        Win32ErrorCodeDescription := 'The password is too complex to be converted to a LAN Manager password. The LAN Manager password returned is a NULL string.';
    Win32ErrorCodes.ERROR_UNKNOWN_REVISION:
        Win32ErrorCodeDescription := 'The revision level is unknown.';
    Win32ErrorCodes.ERROR_REVISION_MISMATCH:
        Win32ErrorCodeDescription := 'Indicates two revision levels are incompatible.';
    Win32ErrorCodes.ERROR_INVALID_OWNER:
        Win32ErrorCodeDescription :=
            'This security ID may not be assigned as the owner of this object.';
    Win32ErrorCodes.ERROR_INVALID_PRIMARY_GROUP:
        Win32ErrorCodeDescription :=
            'This security ID may not be assigned as the primary group of an object.';
    Win32ErrorCodes.ERROR_NO_IMPERSONATION_TOKEN:
        Win32ErrorCodeDescription := 'An attempt has been made to operate on an impersonation token by a thread that is not currently impersonating a client.';
    Win32ErrorCodes.ERROR_CANT_DISABLE_MANDATORY:
        Win32ErrorCodeDescription := 'The group may not be disabled.';
    Win32ErrorCodes.ERROR_NO_LOGON_SERVERS:
        Win32ErrorCodeDescription :=
            'There are currently no logon servers available to service the logon request.';
    Win32ErrorCodes.ERROR_NO_SUCH_LOGON_SESSION:
        Win32ErrorCodeDescription :=
            'A specified logon session does not exist. It may already have been terminated.';
    Win32ErrorCodes.ERROR_NO_SUCH_PRIVILEGE:
        Win32ErrorCodeDescription := 'A specified privilege does not exist.';
    Win32ErrorCodes.ERROR_PRIVILEGE_NOT_HELD:
        Win32ErrorCodeDescription := 'A required privilege is not held by the client.';
    Win32ErrorCodes.ERROR_INVALID_ACCOUNT_NAME:
        Win32ErrorCodeDescription := 'The name provided is not a properly formed account name.';
    Win32ErrorCodes.ERROR_USER_EXISTS:
        Win32ErrorCodeDescription := 'The specified user already exists.';
    Win32ErrorCodes.ERROR_NO_SUCH_USER:
        Win32ErrorCodeDescription := 'The specified user does not exist.';
    Win32ErrorCodes.ERROR_GROUP_EXISTS:
        Win32ErrorCodeDescription := 'The specified group already exists.';
    Win32ErrorCodes.ERROR_NO_SUCH_GROUP:
        Win32ErrorCodeDescription := 'The specified group does not exist.';
    Win32ErrorCodes.ERROR_MEMBER_IN_GROUP:
        Win32ErrorCodeDescription := 'Either the specified user account is already a member of the specified group, or the specified group cannot be deleted because it contains a member.';
    Win32ErrorCodes.ERROR_MEMBER_NOT_IN_GROUP:
        Win32ErrorCodeDescription :=
            'The specified user account is not a member of the specified group account.';
    Win32ErrorCodes.ERROR_LAST_ADMIN:
        Win32ErrorCodeDescription :=
            'The last remaining administration account cannot be disabled or deleted.';
    Win32ErrorCodes.ERROR_WRONG_PASSWORD:
        Win32ErrorCodeDescription :=
            'Unable to update the password. The value provided as the current password is incorrect.';
    Win32ErrorCodes.ERROR_ILL_FORMED_PASSWORD:
        Win32ErrorCodeDescription := 'Unable to update the password. The value provided for the new password contains values that are not allowed in passwords.';
    Win32ErrorCodes.ERROR_PASSWORD_RESTRICTION:
        Win32ErrorCodeDescription := 'Unable to update the password. The value provided for the new password does not meet the length, complexity, or history requirement of the domain.';
    Win32ErrorCodes.ERROR_LOGON_FAILURE:
        Win32ErrorCodeDescription := 'Logon failure: unknown user name or bad password.';
    Win32ErrorCodes.ERROR_ACCOUNT_RESTRICTION:
        Win32ErrorCodeDescription := 'Logon failure: user account restriction.';
    Win32ErrorCodes.ERROR_INVALID_LOGON_HOURS:
        Win32ErrorCodeDescription := 'Logon failure: account logon time restriction violation.';
    Win32ErrorCodes.ERROR_INVALID_WORKSTATION:
        Win32ErrorCodeDescription := 'Logon failure: user not allowed to log on to this computer.';
    Win32ErrorCodes.ERROR_PASSWORD_EXPIRED:
        Win32ErrorCodeDescription := 'Logon failure: the specified account password has expired.';
    Win32ErrorCodes.ERROR_ACCOUNT_DISABLED:
        Win32ErrorCodeDescription := 'Logon failure: account currently disabled.';
    Win32ErrorCodes.ERROR_NONE_MAPPED:
        Win32ErrorCodeDescription := 'No mapping between account names and security IDs was done.';
    Win32ErrorCodes.ERROR_TOO_MANY_LUIDS_REQUESTED:
        Win32ErrorCodeDescription :=
            'Too many local user identifiers (LUIDs) were requested at one time.';
    Win32ErrorCodes.ERROR_LUIDS_EXHAUSTED:
        Win32ErrorCodeDescription := 'No more local user identifiers (LUIDs) are available.';
    Win32ErrorCodes.ERROR_INVALID_SUB_AUTHORITY:
        Win32ErrorCodeDescription :=
            'The subauthority part of a security ID is invalid for this particular use.';
    Win32ErrorCodes.ERROR_INVALID_ACL:
        Win32ErrorCodeDescription := 'The access control list (ACL) structure is invalid.';
    Win32ErrorCodes.ERROR_INVALID_SID:
        Win32ErrorCodeDescription := 'The security ID structure is invalid.';
    Win32ErrorCodes.ERROR_INVALID_SECURITY_DESCR:
        Win32ErrorCodeDescription := 'The security descriptor structure is invalid.';
    Win32ErrorCodes.ERROR_BAD_INHERITANCE_ACL:
        Win32ErrorCodeDescription :=
            'The inherited access control list (ACL) or access control entry (ACE) could not be built.';
    Win32ErrorCodes.ERROR_SERVER_DISABLED:
        Win32ErrorCodeDescription := 'The server is currently disabled.';
    Win32ErrorCodes.ERROR_SERVER_NOT_DISABLED:
        Win32ErrorCodeDescription := 'The server is currently enabled.';
    Win32ErrorCodes.ERROR_INVALID_ID_AUTHORITY:
        Win32ErrorCodeDescription :=
            'The value provided was an invalid value for an identifier authority.';
    Win32ErrorCodes.ERROR_ALLOTTED_SPACE_EXCEEDED:
        Win32ErrorCodeDescription :=
            'No more memory is available for security information updates.';
    Win32ErrorCodes.ERROR_INVALID_GROUP_ATTRIBUTES:
        Win32ErrorCodeDescription := 'The specified attributes are invalid, or incompatible with the attributes for the group as a whole.';
    Win32ErrorCodes.ERROR_BAD_IMPERSONATION_LEVEL:
        Win32ErrorCodeDescription := 'Either a required impersonation level was not provided, or the provided impersonation level is invalid.';
    Win32ErrorCodes.ERROR_CANT_OPEN_ANONYMOUS:
        Win32ErrorCodeDescription := 'Cannot open an anonymous level security token.';
    Win32ErrorCodes.ERROR_BAD_VALIDATION_CLASS:
        Win32ErrorCodeDescription := 'The validation information class requested was invalid.';
    Win32ErrorCodes.ERROR_BAD_TOKEN_TYPE:
        Win32ErrorCodeDescription :=
            'The type of the token is inappropriate for its attempted use.';
    Win32ErrorCodes.ERROR_NO_SECURITY_ON_OBJECT:
        Win32ErrorCodeDescription :=
            'Unable to perform a security operation on an object that has no associated security.';
    Win32ErrorCodes.ERROR_CANT_ACCESS_DOMAIN_INFO:
        Win32ErrorCodeDescription := 'Configuration information could not be read from the domain controller, either because the machine is unavailable, or access has been denied.';
    Win32ErrorCodes.ERROR_INVALID_SERVER_STATE:
        Win32ErrorCodeDescription := 'The security account manager (SAM) or local security authority (LSA) server was in the wrong state to perform the security operation.';
    Win32ErrorCodes.ERROR_INVALID_DOMAIN_STATE:
        Win32ErrorCodeDescription :=
            'The domain was in the wrong state to perform the security operation.';
    Win32ErrorCodes.ERROR_INVALID_DOMAIN_ROLE:
        Win32ErrorCodeDescription :=
            'This operation is only allowed for the Primary Domain Controller of the domain.';
    Win32ErrorCodes.ERROR_NO_SUCH_DOMAIN:
        Win32ErrorCodeDescription :=
            'The specified domain either does not exist or could not be contacted.';
    Win32ErrorCodes.ERROR_DOMAIN_EXISTS:
        Win32ErrorCodeDescription := 'The specified domain already exists.';
    Win32ErrorCodes.ERROR_DOMAIN_LIMIT_EXCEEDED:
        Win32ErrorCodeDescription :=
            'An attempt was made to exceed the limit on the number of domains per server.';
    Win32ErrorCodes.ERROR_INTERNAL_DB_CORRUPTION:
        Win32ErrorCodeDescription := 'Unable to complete the requested operation because of either a catastrophic media failure or a data structure corruption on the disk.';
    Win32ErrorCodes.ERROR_INTERNAL_ERROR:
        Win32ErrorCodeDescription := 'An internal error occurred.';
    Win32ErrorCodes.ERROR_GENERIC_NOT_MAPPED:
        Win32ErrorCodeDescription := 'Generic access types were contained in an access mask which should already be mapped to nongeneric types.';
    Win32ErrorCodes.ERROR_BAD_DESCRIPTOR_FORMAT:
        Win32ErrorCodeDescription :=
            'A security descriptor is not in the right format (absolute or self-relative).';
    Win32ErrorCodes.ERROR_NOT_LOGON_PROCESS:
        Win32ErrorCodeDescription := 'The requested action is restricted for use by logon processes only. The calling process has not registered as a logon process.';
    Win32ErrorCodes.ERROR_LOGON_SESSION_EXISTS:
        Win32ErrorCodeDescription :=
            'Cannot start a new logon session with an ID that is already in use.';
    Win32ErrorCodes.ERROR_NO_SUCH_PACKAGE:
        Win32ErrorCodeDescription := 'A specified authentication package is unknown.';
    Win32ErrorCodes.ERROR_BAD_LOGON_SESSION_STATE:
        Win32ErrorCodeDescription :=
            'The logon session is not in a state that is consistent with the requested operation.';
    Win32ErrorCodes.ERROR_LOGON_SESSION_COLLISION:
        Win32ErrorCodeDescription := 'The logon session ID is already in use.';
    Win32ErrorCodes.ERROR_INVALID_LOGON_TYPE:
        Win32ErrorCodeDescription := 'A logon request contained an invalid logon type value.';
    Win32ErrorCodes.ERROR_CANNOT_IMPERSONATE:
        Win32ErrorCodeDescription :=
            'Unable to impersonate using a named pipe until data has been read from that pipe.';
    Win32ErrorCodes.ERROR_RXACT_INVALID_STATE:
        Win32ErrorCodeDescription :=
            'The transaction state of a registry subtree is incompatible with the requested operation.';
    Win32ErrorCodes.ERROR_RXACT_COMMIT_FAILURE:
        Win32ErrorCodeDescription :=
            'An internal security database corruption has been encountered.';
    Win32ErrorCodes.ERROR_SPECIAL_ACCOUNT:
        Win32ErrorCodeDescription := 'Cannot perform this operation on built-in accounts.';
    Win32ErrorCodes.ERROR_SPECIAL_GROUP:
        Win32ErrorCodeDescription :=
            'Cannot perform this operation on this built-in special group.';
    Win32ErrorCodes.ERROR_SPECIAL_USER:
        Win32ErrorCodeDescription :=
            'Cannot perform this operation on this built-in special user.';
    Win32ErrorCodes.ERROR_MEMBERS_PRIMARY_GROUP:
        Win32ErrorCodeDescription := 'The user cannot be removed from a group because the group is currently the users primary group.';
    Win32ErrorCodes.ERROR_TOKEN_ALREADY_IN_USE:
        Win32ErrorCodeDescription := 'The token is already in use as a primary token.';
    Win32ErrorCodes.ERROR_NO_SUCH_ALIAS:
        Win32ErrorCodeDescription := 'The specified local group does not exist.';
    Win32ErrorCodes.ERROR_MEMBER_NOT_IN_ALIAS:
        Win32ErrorCodeDescription :=
            'The specified account name is not a member of the local group.';
    Win32ErrorCodes.ERROR_MEMBER_IN_ALIAS:
        Win32ErrorCodeDescription :=
            'The specified account name is already a member of the local group.';
    Win32ErrorCodes.ERROR_ALIAS_EXISTS:
        Win32ErrorCodeDescription := 'The specified local group already exists.';
    Win32ErrorCodes.ERROR_LOGON_NOT_GRANTED:
        Win32ErrorCodeDescription :=
            'Logon failure: the user has not been granted the requested logon type at this computer.';
    Win32ErrorCodes.ERROR_TOO_MANY_SECRETS:
        Win32ErrorCodeDescription :=
            'The maximum number of secrets that may be stored in a single system has been exceeded.';
    Win32ErrorCodes.ERROR_SECRET_TOO_LONG:
        Win32ErrorCodeDescription := 'The length of a secret exceeds the maximum length allowed.';
    Win32ErrorCodes.ERROR_INTERNAL_DB_ERROR:
        Win32ErrorCodeDescription :=
            'The local security authority database contains an internal inconsistency.';
    Win32ErrorCodes.ERROR_TOO_MANY_CONTEXT_IDS:
        Win32ErrorCodeDescription :=
            'During a logon attempt, the users security context accumulated too many security IDs.';
    Win32ErrorCodes.ERROR_LOGON_TYPE_NOT_GRANTED:
        Win32ErrorCodeDescription :=
            'Logon failure: the user has not been granted the requested logon type at this computer.';
    Win32ErrorCodes.ERROR_NT_CROSS_ENCRYPTION_REQUIRED:
        Win32ErrorCodeDescription :=
            'A cross-encrypted password is necessary to change a user password.';
    Win32ErrorCodes.ERROR_NO_SUCH_MEMBER:
        Win32ErrorCodeDescription := 'A new member could not be added to or removed from the local group because the member does not exist.';
    Win32ErrorCodes.ERROR_INVALID_MEMBER:
        Win32ErrorCodeDescription := 'A new member could not be added to a local group because the member has the wrong account type.';
    Win32ErrorCodes.ERROR_TOO_MANY_SIDS:
        Win32ErrorCodeDescription := 'Too many security IDs have been specified.';
    Win32ErrorCodes.ERROR_LM_CROSS_ENCRYPTION_REQUIRED:
        Win32ErrorCodeDescription :=
            'A cross-encrypted password is necessary to change this user password.';
    Win32ErrorCodes.ERROR_NO_INHERITANCE:
        Win32ErrorCodeDescription := 'Indicates an ACL contains no inheritable components.';
    Win32ErrorCodes.ERROR_FILE_CORRUPT:
        Win32ErrorCodeDescription := 'The file or directory is corrupted and unreadable.';
    Win32ErrorCodes.ERROR_DISK_CORRUPT:
        Win32ErrorCodeDescription := 'The disk structure is corrupted and unreadable.';
    Win32ErrorCodes.ERROR_NO_USER_SESSION_KEY:
        Win32ErrorCodeDescription :=
            'There is no user session key for the specified logon session.';
    Win32ErrorCodes.ERROR_LICENSE_QUOTA_EXCEEDED:
        Win32ErrorCodeDescription := 'The service being accessed is licensed for a particular number of connections. No more connections can be made to the service at this time because there are already as many connections as the service can accept.';
    Win32ErrorCodes.ERROR_WRONG_TARGET_NAME:
        Win32ErrorCodeDescription := 'Logon Failure: The target account name is incorrect.';
    Win32ErrorCodes.ERROR_MUTUAL_AUTH_FAILED:
        Win32ErrorCodeDescription := 'Mutual Authentication failed. The servers password is out of date at the domain controller.';
    Win32ErrorCodes.ERROR_TIME_SKEW:
        Win32ErrorCodeDescription := 'There is a time difference between the client and server.';
    Win32ErrorCodes.ERROR_CURRENT_DOMAIN_NOT_ALLOWED:
        Win32ErrorCodeDescription := 'This operation can not be performed on the current domain.';
    Win32ErrorCodes.ERROR_INVALID_WINDOW_HANDLE:
        Win32ErrorCodeDescription := 'Invalid window handle.';
    Win32ErrorCodes.ERROR_INVALID_MENU_HANDLE:
        Win32ErrorCodeDescription := 'Invalid menu handle.';
    Win32ErrorCodes.ERROR_INVALID_CURSOR_HANDLE:
        Win32ErrorCodeDescription := 'Invalid cursor handle.';
    Win32ErrorCodes.ERROR_INVALID_ACCEL_HANDLE:
        Win32ErrorCodeDescription := 'Invalid accelerator table handle.';
    Win32ErrorCodes.ERROR_INVALID_HOOK_HANDLE:
        Win32ErrorCodeDescription := 'Invalid hook handle.';
    Win32ErrorCodes.ERROR_INVALID_DWP_HANDLE:
        Win32ErrorCodeDescription := 'Invalid handle to a multiple-window position structure.';
    Win32ErrorCodes.ERROR_TLW_WITH_WSCHILD:
        Win32ErrorCodeDescription := 'Cannot create a top-level child window.';
    Win32ErrorCodes.ERROR_CANNOT_FIND_WND_CLASS:
        Win32ErrorCodeDescription := 'Cannot find window class.';
    Win32ErrorCodes.ERROR_WINDOW_OF_OTHER_THREAD:
        Win32ErrorCodeDescription := 'Invalid window; it belongs to other thread.';
    Win32ErrorCodes.ERROR_HOTKEY_ALREADY_REGISTERED:
        Win32ErrorCodeDescription := 'Hot key is already registered.';
    Win32ErrorCodes.ERROR_CLASS_ALREADY_EXISTS:
        Win32ErrorCodeDescription := 'Class already exists.';
    Win32ErrorCodes.ERROR_CLASS_DOES_NOT_EXIST:
        Win32ErrorCodeDescription := 'Class does not exist.';
    Win32ErrorCodes.ERROR_CLASS_HAS_WINDOWS:
        Win32ErrorCodeDescription := 'Class still has open windows.';
    Win32ErrorCodes.ERROR_INVALID_INDEX:
        Win32ErrorCodeDescription := 'Invalid index.';
    Win32ErrorCodes.ERROR_INVALID_ICON_HANDLE:
        Win32ErrorCodeDescription := 'Invalid icon handle.';
    Win32ErrorCodes.ERROR_PRIVATE_DIALOG_INDEX:
        Win32ErrorCodeDescription := 'Using private DIALOG window words.';
    Win32ErrorCodes.ERROR_LISTBOX_ID_NOT_FOUND:
        Win32ErrorCodeDescription := 'The list box identifier was not found.';
    Win32ErrorCodes.ERROR_NO_WILDCARD_CHARACTERS:
        Win32ErrorCodeDescription := 'No wildcards were found.';
    Win32ErrorCodes.ERROR_CLIPBOARD_NOT_OPEN:
        Win32ErrorCodeDescription := 'Thread does not have a clipboard open.';
    Win32ErrorCodes.ERROR_HOTKEY_NOT_REGISTERED:
        Win32ErrorCodeDescription := 'Hot key is not registered.';
    Win32ErrorCodes.ERROR_WINDOW_NOT_DIALOG:
        Win32ErrorCodeDescription := 'The window is not a valid dialog window.';
    Win32ErrorCodes.ERROR_CONTROL_ID_NOT_FOUND:
        Win32ErrorCodeDescription := 'Control ID not found.';
    Win32ErrorCodes.ERROR_INVALID_COMBOBOX_MESSAGE:
        Win32ErrorCodeDescription :=
            'Invalid message for a combo box because it does not have an edit control.';
    Win32ErrorCodes.ERROR_WINDOW_NOT_COMBOBOX:
        Win32ErrorCodeDescription := 'The window is not a combo box.';
    Win32ErrorCodes.ERROR_INVALID_EDIT_HEIGHT:
        Win32ErrorCodeDescription := 'Height must be less than 256.';
    Win32ErrorCodes.ERROR_DC_NOT_FOUND:
        Win32ErrorCodeDescription := 'Invalid device context (DC) handle.';
    Win32ErrorCodes.ERROR_INVALID_HOOK_FILTER:
        Win32ErrorCodeDescription := 'Invalid hook procedure type.';
    Win32ErrorCodes.ERROR_INVALID_FILTER_PROC:
        Win32ErrorCodeDescription := 'Invalid hook procedure.';
    Win32ErrorCodes.ERROR_HOOK_NEEDS_HMOD:
        Win32ErrorCodeDescription := 'Cannot set nonlocal hook without a module handle.';
    Win32ErrorCodes.ERROR_GLOBAL_ONLY_HOOK:
        Win32ErrorCodeDescription := 'This hook procedure can only be set globally.';
    Win32ErrorCodes.ERROR_JOURNAL_HOOK_SET:
        Win32ErrorCodeDescription := 'The journal hook procedure is already installed.';
    Win32ErrorCodes.ERROR_HOOK_NOT_INSTALLED:
        Win32ErrorCodeDescription := 'The hook procedure is not installed.';
    Win32ErrorCodes.ERROR_INVALID_LB_MESSAGE:
        Win32ErrorCodeDescription := 'Invalid message for single-selection list box.';
    Win32ErrorCodes.ERROR_SETCOUNT_ON_BAD_LB:
        Win32ErrorCodeDescription := 'LB_SETCOUNT sent to non-lazy list box.';
    Win32ErrorCodes.ERROR_LB_WITHOUT_TABSTOPS:
        Win32ErrorCodeDescription := 'This list box does not support tab stops.';
    Win32ErrorCodes.ERROR_DESTROY_OBJECT_OF_OTHER_THREAD:
        Win32ErrorCodeDescription := 'Cannot destroy object created by another thread.';
    Win32ErrorCodes.ERROR_CHILD_WINDOW_MENU:
        Win32ErrorCodeDescription := 'Child windows cannot have menus.';
    Win32ErrorCodes.ERROR_NO_SYSTEM_MENU:
        Win32ErrorCodeDescription := 'The window does not have a system menu.';
    Win32ErrorCodes.ERROR_INVALID_MSGBOX_STYLE:
        Win32ErrorCodeDescription := 'Invalid message box style.';
    Win32ErrorCodes.ERROR_INVALID_SPI_VALUE:
        Win32ErrorCodeDescription := 'Invalid system-wide (SPI_*) parameter.';
    Win32ErrorCodes.ERROR_SCREEN_ALREADY_LOCKED:
        Win32ErrorCodeDescription := 'Screen already locked.';
    Win32ErrorCodes.ERROR_HWNDS_HAVE_DIFF_PARENT:
        Win32ErrorCodeDescription :=
            'All handles to windows in a multiple-window position structure must have the same parent.';
    Win32ErrorCodes.ERROR_NOT_CHILD_WINDOW:
        Win32ErrorCodeDescription := 'The window is not a child window.';
    Win32ErrorCodes.ERROR_INVALID_GW_COMMAND:
        Win32ErrorCodeDescription := 'Invalid GW_* command.';
    Win32ErrorCodes.ERROR_INVALID_THREAD_ID:
        Win32ErrorCodeDescription := 'Invalid thread identifier.';
    Win32ErrorCodes.ERROR_NON_MDICHILD_WINDOW:
        Win32ErrorCodeDescription := 'Cannot process a message from a window that is not a multiple document interface (MDI) window.';
    Win32ErrorCodes.ERROR_POPUP_ALREADY_ACTIVE:
        Win32ErrorCodeDescription := 'Popup menu already active.';
    Win32ErrorCodes.ERROR_NO_SCROLLBARS:
        Win32ErrorCodeDescription := 'The window does not have scroll bars.';
    Win32ErrorCodes.ERROR_INVALID_SCROLLBAR_RANGE:
        Win32ErrorCodeDescription := 'Scroll bar range cannot be greater than MAXLONG.';
    Win32ErrorCodes.ERROR_INVALID_SHOWWIN_COMMAND:
        Win32ErrorCodeDescription := 'Cannot show or remove the window in the way specified.';
    Win32ErrorCodes.ERROR_NO_SYSTEM_RESOURCES:
        Win32ErrorCodeDescription :=
            'Insufficient system resources exist to complete the requested service.';
    Win32ErrorCodes.ERROR_NONPAGED_SYSTEM_RESOURCES:
        Win32ErrorCodeDescription :=
            'Insufficient system resources exist to complete the requested service.';
    Win32ErrorCodes.ERROR_PAGED_SYSTEM_RESOURCES:
        Win32ErrorCodeDescription :=
            'Insufficient system resources exist to complete the requested service.';
    Win32ErrorCodes.ERROR_WORKING_SET_QUOTA:
        Win32ErrorCodeDescription := 'Insufficient quota to complete the requested service.';
    Win32ErrorCodes.ERROR_PAGEFILE_QUOTA:
        Win32ErrorCodeDescription := 'Insufficient quota to complete the requested service.';
    Win32ErrorCodes.ERROR_COMMITMENT_LIMIT:
        Win32ErrorCodeDescription :=
            'The paging file is too small for this operation to complete.';
    Win32ErrorCodes.ERROR_MENU_ITEM_NOT_FOUND:
        Win32ErrorCodeDescription := 'A menu item was not found.';
    Win32ErrorCodes.ERROR_INVALID_KEYBOARD_HANDLE:
        Win32ErrorCodeDescription := 'Invalid keyboard layout handle.';
    Win32ErrorCodes.ERROR_HOOK_TYPE_NOT_ALLOWED:
        Win32ErrorCodeDescription := 'Hook type not allowed.';
    Win32ErrorCodes.ERROR_REQUIRES_INTERACTIVE_WINDOWSTATION:
        Win32ErrorCodeDescription := 'This operation requires an interactive window station.';
    Win32ErrorCodes.ERROR_TIMEOUT:
        Win32ErrorCodeDescription := 'This operation returned because the timeout period expired.';
    Win32ErrorCodes.ERROR_INVALID_MONITOR_HANDLE:
        Win32ErrorCodeDescription := 'Invalid monitor handle.';
    Win32ErrorCodes.ERROR_EVENTLOG_FILE_CORRUPT:
        Win32ErrorCodeDescription := 'The event log file is corrupted.';
    Win32ErrorCodes.ERROR_EVENTLOG_CANT_START:
        Win32ErrorCodeDescription :=
            'No event log file could be opened, so the event logging service did not start.';
    Win32ErrorCodes.ERROR_LOG_FILE_FULL:
        Win32ErrorCodeDescription := 'The event log file is full.';
    Win32ErrorCodes.ERROR_EVENTLOG_FILE_CHANGED:
        Win32ErrorCodeDescription := 'The event log file has changed between read operations.';
    Win32ErrorCodes.ERROR_INSTALL_SERVICE_FAILURE:
        Win32ErrorCodeDescription := 'The Windows Installer service could not be accessed. Contact your support personnel to verify that the Windows Installer service is properly registered.';
    Win32ErrorCodes.ERROR_INSTALL_USEREXIT:
        Win32ErrorCodeDescription := 'User cancelled installation.';
    Win32ErrorCodes.ERROR_INSTALL_FAILURE:
        Win32ErrorCodeDescription := 'Fatal error during installation.';
    Win32ErrorCodes.ERROR_INSTALL_SUSPEND:
        Win32ErrorCodeDescription := 'Installation suspended, incomplete.';
    Win32ErrorCodes.ERROR_UNKNOWN_PRODUCT:
        Win32ErrorCodeDescription :=
            'This action is only valid for products that are currently installed.';
    Win32ErrorCodes.ERROR_UNKNOWN_FEATURE:
        Win32ErrorCodeDescription := 'Feature ID not registered.';
    Win32ErrorCodes.ERROR_UNKNOWN_COMPONENT:
        Win32ErrorCodeDescription := 'Component ID not registered.';
    Win32ErrorCodes.ERROR_UNKNOWN_PROPERTY:
        Win32ErrorCodeDescription := 'Unknown property.';
    Win32ErrorCodes.ERROR_INVALID_HANDLE_STATE:
        Win32ErrorCodeDescription := 'Handle is in an invalid state.';
    Win32ErrorCodes.ERROR_BAD_CONFIGURATION:
        Win32ErrorCodeDescription :=
            'The configuration data for this product is corrupt. Contact your support personnel.';
    Win32ErrorCodes.ERROR_INDEX_ABSENT:
        Win32ErrorCodeDescription := 'Component qualifier not present.';
    Win32ErrorCodes.ERROR_INSTALL_SOURCE_ABSENT:
        Win32ErrorCodeDescription := 'The installation source for this product is not available. Verify that the source exists and that you can access it.';
    Win32ErrorCodes.ERROR_INSTALL_PACKAGE_VERSION:
        Win32ErrorCodeDescription := 'This installation package cannot be installed by the Windows Installer service. You must install a Windows service pack that contains a newer version of the Windows Installer service.';
    Win32ErrorCodes.ERROR_PRODUCT_UNINSTALLED:
        Win32ErrorCodeDescription := 'Product is uninstalled.';
    Win32ErrorCodes.ERROR_BAD_QUERY_SYNTAX:
        Win32ErrorCodeDescription := 'SQL query syntax invalid or unsupported.';
    Win32ErrorCodes.ERROR_INVALID_FIELD:
        Win32ErrorCodeDescription := 'Record field does not exist.';
    Win32ErrorCodes.ERROR_DEVICE_REMOVED:
        Win32ErrorCodeDescription := 'The device has been removed.';
    Win32ErrorCodes.ERROR_INSTALL_ALREADY_RUNNING:
        Win32ErrorCodeDescription := 'Another installation is already in progress. Complete that installation before proceeding with this install.';
    Win32ErrorCodes.ERROR_INSTALL_PACKAGE_OPEN_FAILED:
        Win32ErrorCodeDescription := 'This installation package could not be opened. Verify that the package exists and that you can access it, or contact the application vendor to verify that this is a valid Windows Installer package.';
    Win32ErrorCodes.ERROR_INSTALL_PACKAGE_INVALID:
        Win32ErrorCodeDescription := 'This installation package could not be opened. Contact the application vendor to verify that this is a valid Windows Installer package.';
    Win32ErrorCodes.ERROR_INSTALL_UI_FAILURE:
        Win32ErrorCodeDescription := 'There was an error starting the Windows Installer service user interface. Contact your support personnel.';
    Win32ErrorCodes.ERROR_INSTALL_LOG_FAILURE:
        Win32ErrorCodeDescription := 'Error opening installation log file. Verify that the specified log file location exists and that you can write to it.';
    Win32ErrorCodes.ERROR_INSTALL_LANGUAGE_UNSUPPORTED:
        Win32ErrorCodeDescription :=
            'The language of this installation package is not supported by your system.';
    Win32ErrorCodes.ERROR_INSTALL_TRANSFORM_FAILURE:
        Win32ErrorCodeDescription :=
            'Error applying transforms. Verify that the specified transform paths are valid.';
    Win32ErrorCodes.ERROR_INSTALL_PACKAGE_REJECTED:
        Win32ErrorCodeDescription :=
            'This installation is forbidden by system policy. Contact your system administrator.';
    Win32ErrorCodes.ERROR_FUNCTION_NOT_CALLED:
        Win32ErrorCodeDescription := 'Function could not be executed.';
    Win32ErrorCodes.ERROR_FUNCTION_FAILED:
        Win32ErrorCodeDescription := 'Function failed during execution.';
    Win32ErrorCodes.ERROR_INVALID_TABLE:
        Win32ErrorCodeDescription := 'Invalid or unknown table specified.';
    Win32ErrorCodes.ERROR_DATATYPE_MISMATCH:
        Win32ErrorCodeDescription := 'Data supplied is of wrong type.';
    Win32ErrorCodes.ERROR_UNSUPPORTED_TYPE:
        Win32ErrorCodeDescription := 'Data of this type is not supported.';
    Win32ErrorCodes.ERROR_CREATE_FAILED:
        Win32ErrorCodeDescription :=
            'The Windows Installer service failed to start. Contact your support personnel.';
    Win32ErrorCodes.ERROR_INSTALL_TEMP_UNWRITABLE:
        Win32ErrorCodeDescription := 'The temp folder is either full or inaccessible. Verify that the temp folder exists and that you can write to it.';
    Win32ErrorCodes.ERROR_INSTALL_PLATFORM_UNSUPPORTED:
        Win32ErrorCodeDescription := 'This installation package is not supported by this processor type. Contact your product vendor.';
    Win32ErrorCodes.ERROR_INSTALL_NOTUSED:
        Win32ErrorCodeDescription := 'Component not used on this computer.';
    Win32ErrorCodes.ERROR_PATCH_PACKAGE_OPEN_FAILED:
        Win32ErrorCodeDescription := 'This patch package could not be opened. Verify that the patch package exists and that you can access it, or contact the application vendor to verify that this is a valid Windows Installer patch package.';
    Win32ErrorCodes.ERROR_PATCH_PACKAGE_INVALID:
        Win32ErrorCodeDescription := 'This patch package could not be opened. Contact the application vendor to verify that this is a valid Windows Installer patch package.';
    Win32ErrorCodes.ERROR_PATCH_PACKAGE_UNSUPPORTED:
        Win32ErrorCodeDescription := 'This patch package cannot be processed by the Windows Installer service. You must install a Windows service pack that contains a newer version of the Windows Installer service.';
    Win32ErrorCodes.ERROR_PRODUCT_VERSION:
        Win32ErrorCodeDescription := 'Another version of this product is already installed. Installation of this version cannot continue. To configure or remove the existing version of this product, use Add/Remove Programs on the Control Panel.';
    Win32ErrorCodes.ERROR_INVALID_COMMAND_LINE:
        Win32ErrorCodeDescription := 'Invalid command line argument. Consult the Windows Installer SDK for detailed command line help.';
    Win32ErrorCodes.ERROR_INSTALL_REMOTE_DISALLOWED:
        Win32ErrorCodeDescription := 'Only administrators have permission to add, remove, or configure server software during a Terminal Services remote session. If you want to install or configure software on the server, contact your network administrator.';
    Win32ErrorCodes.ERROR_SUCCESS_REBOOT_INITIATED:
        Win32ErrorCodeDescription := 'The requested operation completed successfully. The system will be restarted so the changes can take effect.';
    Win32ErrorCodes.ERROR_PATCH_TARGET_NOT_FOUND:
        Win32ErrorCodeDescription := 'The upgrade patch cannot be installed by the Windows Installer service because the program to be upgraded may be missing, or the upgrade patch may update a different version of the program. ';
    Win32ErrorCodes.ERROR_PATCH_PACKAGE_REJECTED:
        Win32ErrorCodeDescription := 'The patch package is not permitted by system policy. It is not signed with an appropriate certificate.';
    Win32ErrorCodes.ERROR_INSTALL_TRANSFORM_REJECTED:
        Win32ErrorCodeDescription := 'One or more customizations are not permitted by system policy. They are not signed with an appropriate certificate.';
    Win32ErrorCodes.RPC_S_INVALID_STRING_BINDING:
        Win32ErrorCodeDescription := 'The string binding is invalid.';
    Win32ErrorCodes.RPC_S_WRONG_KIND_OF_BINDING:
        Win32ErrorCodeDescription := 'The binding handle is not the correct type.';
    Win32ErrorCodes.RPC_S_INVALID_BINDING:
        Win32ErrorCodeDescription := 'The binding handle is invalid.';
    Win32ErrorCodes.RPC_S_PROTSEQ_NOT_SUPPORTED:
        Win32ErrorCodeDescription := 'The RPC protocol sequence is not supported.';
    Win32ErrorCodes.RPC_S_INVALID_RPC_PROTSEQ:
        Win32ErrorCodeDescription := 'The RPC protocol sequence is invalid.';
    Win32ErrorCodes.RPC_S_INVALID_STRING_UUID:
        Win32ErrorCodeDescription := 'The string universal unique identifier (UUID) is invalid.';
    Win32ErrorCodes.RPC_S_INVALID_ENDPOINT_FORMAT:
        Win32ErrorCodeDescription := 'The endpoint format is invalid.';
    Win32ErrorCodes.RPC_S_INVALID_NET_ADDR:
        Win32ErrorCodeDescription := 'The network address is invalid.';
    Win32ErrorCodes.RPC_S_NO_ENDPOINT_FOUND:
        Win32ErrorCodeDescription := 'No endpoint was found.';
    Win32ErrorCodes.RPC_S_INVALID_TIMEOUT:
        Win32ErrorCodeDescription := 'The timeout value is invalid.';
    Win32ErrorCodes.RPC_S_OBJECT_NOT_FOUND:
        Win32ErrorCodeDescription :=
            'The object universal unique identifier (UUID) was not found.';
    Win32ErrorCodes.RPC_S_ALREADY_REGISTERED:
        Win32ErrorCodeDescription :=
            'The object universal unique identifier (UUID) has already been registered.';
    Win32ErrorCodes.RPC_S_TYPE_ALREADY_REGISTERED:
        Win32ErrorCodeDescription :=
            'The type universal unique identifier (UUID) has already been registered.';
    Win32ErrorCodes.RPC_S_ALREADY_LISTENING:
        Win32ErrorCodeDescription := 'The RPC server is already listening.';
    Win32ErrorCodes.RPC_S_NO_PROTSEQS_REGISTERED:
        Win32ErrorCodeDescription := 'No protocol sequences have been registered.';
    Win32ErrorCodes.RPC_S_NOT_LISTENING:
        Win32ErrorCodeDescription := 'The RPC server is not listening.';
    Win32ErrorCodes.RPC_S_UNKNOWN_MGR_TYPE:
        Win32ErrorCodeDescription := 'The manager type is unknown.';
    Win32ErrorCodes.RPC_S_UNKNOWN_IF:
        Win32ErrorCodeDescription := 'The interface is unknown.';
    Win32ErrorCodes.RPC_S_NO_BINDINGS:
        Win32ErrorCodeDescription := 'There are no bindings.';
    Win32ErrorCodes.RPC_S_NO_PROTSEQS:
        Win32ErrorCodeDescription := 'There are no protocol sequences.';
    Win32ErrorCodes.RPC_S_CANT_CREATE_ENDPOINT:
        Win32ErrorCodeDescription := 'The endpoint cannot be created.';
    Win32ErrorCodes.RPC_S_OUT_OF_RESOURCES:
        Win32ErrorCodeDescription :=
            'Not enough resources are available to complete this operation.';
    Win32ErrorCodes.RPC_S_SERVER_UNAVAILABLE:
        Win32ErrorCodeDescription := 'The RPC server is unavailable.';
    Win32ErrorCodes.RPC_S_SERVER_TOO_BUSY:
        Win32ErrorCodeDescription := 'The RPC server is too busy to complete this operation.';
    Win32ErrorCodes.RPC_S_INVALID_NETWORK_OPTIONS:
        Win32ErrorCodeDescription := 'The network options are invalid.';
    Win32ErrorCodes.RPC_S_NO_CALL_ACTIVE:
        Win32ErrorCodeDescription := 'There are no remote procedure calls active on this thread.';
    Win32ErrorCodes.RPC_S_CALL_FAILED:
        Win32ErrorCodeDescription := 'The remote procedure call failed.';
    Win32ErrorCodes.RPC_S_CALL_FAILED_DNE:
        Win32ErrorCodeDescription := 'The remote procedure call failed and did not execute.';
    Win32ErrorCodes.RPC_S_PROTOCOL_ERROR:
        Win32ErrorCodeDescription := 'A remote procedure call (RPC) protocol error occurred.';
    Win32ErrorCodes.RPC_S_UNSUPPORTED_TRANS_SYN:
        Win32ErrorCodeDescription := 'The transfer syntax is not supported by the RPC server.';
    Win32ErrorCodes.RPC_S_UNSUPPORTED_TYPE:
        Win32ErrorCodeDescription :=
            'The universal unique identifier (UUID) type is not supported.';
    Win32ErrorCodes.RPC_S_INVALID_TAG:
        Win32ErrorCodeDescription := 'The tag is invalid.';
    Win32ErrorCodes.RPC_S_INVALID_BOUND:
        Win32ErrorCodeDescription := 'The array bounds are invalid.';
    Win32ErrorCodes.RPC_S_NO_ENTRY_NAME:
        Win32ErrorCodeDescription := 'The binding does not contain an entry name.';
    Win32ErrorCodes.RPC_S_INVALID_NAME_SYNTAX:
        Win32ErrorCodeDescription := 'The name syntax is invalid.';
    Win32ErrorCodes.RPC_S_UNSUPPORTED_NAME_SYNTAX:
        Win32ErrorCodeDescription := 'The name syntax is not supported.';
    Win32ErrorCodes.RPC_S_UUID_NO_ADDRESS:
        Win32ErrorCodeDescription :=
            'No network address is available to use to construct a universal unique identifier (UUID).';
    Win32ErrorCodes.RPC_S_DUPLICATE_ENDPOINT:
        Win32ErrorCodeDescription := 'The endpoint is a duplicate.';
    Win32ErrorCodes.RPC_S_UNKNOWN_AUTHN_TYPE:
        Win32ErrorCodeDescription := 'The authentication type is unknown.';
    Win32ErrorCodes.RPC_S_MAX_CALLS_TOO_SMALL:
        Win32ErrorCodeDescription := 'The maximum number of calls is too small.';
    Win32ErrorCodes.RPC_S_STRING_TOO_LONG:
        Win32ErrorCodeDescription := 'The string is too long.';
    Win32ErrorCodes.RPC_S_PROTSEQ_NOT_FOUND:
        Win32ErrorCodeDescription := 'The RPC protocol sequence was not found.';
    Win32ErrorCodes.RPC_S_PROCNUM_OUT_OF_RANGE:
        Win32ErrorCodeDescription := 'The procedure number is out of range.';
    Win32ErrorCodes.RPC_S_BINDING_HAS_NO_AUTH:
        Win32ErrorCodeDescription :=
            'The binding does not contain any authentication information.';
    Win32ErrorCodes.RPC_S_UNKNOWN_AUTHN_SERVICE:
        Win32ErrorCodeDescription := 'The authentication service is unknown.';
    Win32ErrorCodes.RPC_S_UNKNOWN_AUTHN_LEVEL:
        Win32ErrorCodeDescription := 'The authentication level is unknown.';
    Win32ErrorCodes.RPC_S_INVALID_AUTH_IDENTITY:
        Win32ErrorCodeDescription := 'The security context is invalid.';
    Win32ErrorCodes.RPC_S_UNKNOWN_AUTHZ_SERVICE:
        Win32ErrorCodeDescription := 'The authorization service is unknown.';
    Win32ErrorCodes.EPT_S_INVALID_ENTRY:
        Win32ErrorCodeDescription := 'The entry is invalid.';
    Win32ErrorCodes.EPT_S_CANT_PERFORM_OP:
        Win32ErrorCodeDescription := 'The server endpoint cannot perform the operation.';
    Win32ErrorCodes.EPT_S_NOT_REGISTERED:
        Win32ErrorCodeDescription :=
            'There are no more endpoints available from the endpoint mapper.';
    Win32ErrorCodes.RPC_S_NOTHING_TO_EXPORT:
        Win32ErrorCodeDescription := 'No interfaces have been exported.';
    Win32ErrorCodes.RPC_S_INCOMPLETE_NAME:
        Win32ErrorCodeDescription := 'The entry name is incomplete.';
    Win32ErrorCodes.RPC_S_INVALID_VERS_OPTION:
        Win32ErrorCodeDescription := 'The version option is invalid.';
    Win32ErrorCodes.RPC_S_NO_MORE_MEMBERS:
        Win32ErrorCodeDescription := 'There are no more members.';
    Win32ErrorCodes.RPC_S_NOT_ALL_OBJS_UNEXPORTED:
        Win32ErrorCodeDescription := 'There is nothing to unexport.';
    Win32ErrorCodes.RPC_S_INTERFACE_NOT_FOUND:
        Win32ErrorCodeDescription := 'The interface was not found.';
    Win32ErrorCodes.RPC_S_ENTRY_ALREADY_EXISTS:
        Win32ErrorCodeDescription := 'The entry already exists.';
    Win32ErrorCodes.RPC_S_ENTRY_NOT_FOUND:
        Win32ErrorCodeDescription := 'The entry is not found.';
    Win32ErrorCodes.RPC_S_NAME_SERVICE_UNAVAILABLE:
        Win32ErrorCodeDescription := 'The name service is unavailable.';
    Win32ErrorCodes.RPC_S_INVALID_NAF_ID:
        Win32ErrorCodeDescription := 'The network address family is invalid.';
    Win32ErrorCodes.RPC_S_CANNOT_SUPPORT:
        Win32ErrorCodeDescription := 'The requested operation is not supported.';
    Win32ErrorCodes.RPC_S_NO_CONTEXT_AVAILABLE:
        Win32ErrorCodeDescription := 'No security context is available to allow impersonation.';
    Win32ErrorCodes.RPC_S_INTERNAL_ERROR:
        Win32ErrorCodeDescription :=
            'An internal error occurred in a remote procedure call (RPC).';
    Win32ErrorCodes.RPC_S_ZERO_DIVIDE:
        Win32ErrorCodeDescription := 'The RPC server attempted an integer division by zero.';
    Win32ErrorCodes.RPC_S_ADDRESS_ERROR:
        Win32ErrorCodeDescription := 'An addressing error occurred in the RPC server.';
    Win32ErrorCodes.RPC_S_FP_DIV_ZERO:
        Win32ErrorCodeDescription :=
            'A floating-point operation at the RPC server caused a division by zero.';
    Win32ErrorCodes.RPC_S_FP_UNDERFLOW:
        Win32ErrorCodeDescription := 'A floating-point underflow occurred at the RPC server.';
    Win32ErrorCodes.RPC_S_FP_OVERFLOW:
        Win32ErrorCodeDescription := 'A floating-point overflow occurred at the RPC server.';
    Win32ErrorCodes.RPC_X_NO_MORE_ENTRIES:
        Win32ErrorCodeDescription :=
            'The list of RPC servers available for the binding of auto handles has been exhausted.';
    Win32ErrorCodes.RPC_X_SS_CHAR_TRANS_OPEN_FAIL:
        Win32ErrorCodeDescription := 'Unable to open the character translation table file.';
    Win32ErrorCodes.RPC_X_SS_CHAR_TRANS_SHORT_FILE:
        Win32ErrorCodeDescription :=
            'The file containing the character translation table has fewer than 512 bytes.';
    Win32ErrorCodes.RPC_X_SS_IN_NULL_CONTEXT:
        Win32ErrorCodeDescription := 'A null context handle was passed from the client to the host during a remote procedure call.';
    Win32ErrorCodes.RPC_X_SS_CONTEXT_DAMAGED:
        Win32ErrorCodeDescription := 'The context handle changed during a remote procedure call.';
    Win32ErrorCodes.RPC_X_SS_HANDLES_MISMATCH:
        Win32ErrorCodeDescription :=
            'The binding handles passed to a remote procedure call do not match.';
    Win32ErrorCodes.RPC_X_SS_CANNOT_GET_CALL_HANDLE:
        Win32ErrorCodeDescription := 'The stub is unable to get the remote procedure call handle.';
    Win32ErrorCodes.RPC_X_NULL_REF_POINTER:
        Win32ErrorCodeDescription := 'A null reference pointer was passed to the stub.';
    Win32ErrorCodes.RPC_X_ENUM_VALUE_OUT_OF_RANGE:
        Win32ErrorCodeDescription := 'The enumeration value is out of range.';
    Win32ErrorCodes.RPC_X_BYTE_COUNT_TOO_SMALL:
        Win32ErrorCodeDescription := 'The byte count is too small.';
    Win32ErrorCodes.RPC_X_BAD_STUB_DATA:
        Win32ErrorCodeDescription := 'The stub received bad data.';
    Win32ErrorCodes.ERROR_INVALID_USER_BUFFER:
        Win32ErrorCodeDescription :=
            'The supplied user buffer is not valid for the requested operation.';
    Win32ErrorCodes.ERROR_UNRECOGNIZED_MEDIA:
        Win32ErrorCodeDescription := 'The disk media is not recognized. It may not be formatted.';
    Win32ErrorCodes.ERROR_NO_TRUST_LSA_SECRET:
        Win32ErrorCodeDescription := 'The workstation does not have a trust secret.';
    Win32ErrorCodes.ERROR_NO_TRUST_SAM_ACCOUNT:
        Win32ErrorCodeDescription := 'The security database on the server does not have a computer account for this workstation trust relationship.';
    Win32ErrorCodes.ERROR_TRUSTED_DOMAIN_FAILURE:
        Win32ErrorCodeDescription :=
            'The trust relationship between the primary domain and the trusted domain failed.';
    Win32ErrorCodes.ERROR_TRUSTED_RELATIONSHIP_FAILURE:
        Win32ErrorCodeDescription :=
            'The trust relationship between this workstation and the primary domain failed.';
    Win32ErrorCodes.ERROR_TRUST_FAILURE:
        Win32ErrorCodeDescription := 'The network logon failed.';
    Win32ErrorCodes.RPC_S_CALL_IN_PROGRESS:
        Win32ErrorCodeDescription :=
            'A remote procedure call is already in progress for this thread.';
    Win32ErrorCodes.ERROR_NETLOGON_NOT_STARTED:
        Win32ErrorCodeDescription :=
            'An attempt was made to logon, but the network logon service was not started.';
    Win32ErrorCodes.ERROR_ACCOUNT_EXPIRED:
        Win32ErrorCodeDescription := 'The users account has expired.';
    Win32ErrorCodes.ERROR_REDIRECTOR_HAS_OPEN_HANDLES:
        Win32ErrorCodeDescription := 'The redirector is in use and cannot be unloaded.';
    Win32ErrorCodes.ERROR_PRINTER_DRIVER_ALREADY_INSTALLED:
        Win32ErrorCodeDescription := 'The specified printer driver is already installed.';
    Win32ErrorCodes.ERROR_UNKNOWN_PORT:
        Win32ErrorCodeDescription := 'The specified port is unknown.';
    Win32ErrorCodes.ERROR_UNKNOWN_PRINTER_DRIVER:
        Win32ErrorCodeDescription := 'The printer driver is unknown.';
    Win32ErrorCodes.ERROR_UNKNOWN_PRINTPROCESSOR:
        Win32ErrorCodeDescription := 'The print processor is unknown.';
    Win32ErrorCodes.ERROR_INVALID_SEPARATOR_FILE:
        Win32ErrorCodeDescription := 'The specified separator file is invalid.';
    Win32ErrorCodes.ERROR_INVALID_PRIORITY:
        Win32ErrorCodeDescription := 'The specified priority is invalid.';
    Win32ErrorCodes.ERROR_INVALID_PRINTER_NAME:
        Win32ErrorCodeDescription := 'The printer name is invalid.';
    Win32ErrorCodes.ERROR_PRINTER_ALREADY_EXISTS:
        Win32ErrorCodeDescription := 'The printer already exists.';
    Win32ErrorCodes.ERROR_INVALID_PRINTER_COMMAND:
        Win32ErrorCodeDescription := 'The printer command is invalid.';
    Win32ErrorCodes.ERROR_INVALID_DATATYPE:
        Win32ErrorCodeDescription := 'The specified datatype is invalid.';
    Win32ErrorCodes.ERROR_INVALID_ENVIRONMENT:
        Win32ErrorCodeDescription := 'The environment specified is invalid.';
    Win32ErrorCodes.RPC_S_NO_MORE_BINDINGS:
        Win32ErrorCodeDescription := 'There are no more bindings.';
    Win32ErrorCodes.ERROR_NOLOGON_INTERDOMAIN_TRUST_ACCOUNT:
        Win32ErrorCodeDescription := 'The account used is an interdomain trust account. Use your global user account or local user account to access this server.';
    Win32ErrorCodes.ERROR_NOLOGON_WORKSTATION_TRUST_ACCOUNT:
        Win32ErrorCodeDescription := 'The account used is a computer account. Use your global user account or local user account to access this server.';
    Win32ErrorCodes.ERROR_NOLOGON_SERVER_TRUST_ACCOUNT:
        Win32ErrorCodeDescription := 'The account used is a server trust account. Use your global user account or local user account to access this server.';
    Win32ErrorCodes.ERROR_DOMAIN_TRUST_INCONSISTENT:
        Win32ErrorCodeDescription := 'The name or security ID (SID) of the domain specified is inconsistent with the trust information for that domain.';
    Win32ErrorCodes.ERROR_SERVER_HAS_OPEN_HANDLES:
        Win32ErrorCodeDescription := 'The server is in use and cannot be unloaded.';
    Win32ErrorCodes.ERROR_RESOURCE_DATA_NOT_FOUND:
        Win32ErrorCodeDescription :=
            'The specified image file did not contain a resource section.';
    Win32ErrorCodes.ERROR_RESOURCE_TYPE_NOT_FOUND:
        Win32ErrorCodeDescription :=
            'The specified resource type cannot be found in the image file.';
    Win32ErrorCodes.ERROR_RESOURCE_NAME_NOT_FOUND:
        Win32ErrorCodeDescription :=
            'The specified resource name cannot be found in the image file.';
    Win32ErrorCodes.ERROR_RESOURCE_LANG_NOT_FOUND:
        Win32ErrorCodeDescription :=
            'The specified resource language ID cannot be found in the image file.';
    Win32ErrorCodes.ERROR_NOT_ENOUGH_QUOTA:
        Win32ErrorCodeDescription := 'Not enough quota is available to process this command.';
    Win32ErrorCodes.RPC_S_NO_INTERFACES:
        Win32ErrorCodeDescription := 'No interfaces have been registered.';
    Win32ErrorCodes.RPC_S_CALL_CANCELLED:
        Win32ErrorCodeDescription := 'The remote procedure call was cancelled.';
    Win32ErrorCodes.RPC_S_BINDING_INCOMPLETE:
        Win32ErrorCodeDescription :=
            'The binding handle does not contain all required information.';
    Win32ErrorCodes.RPC_S_COMM_FAILURE:
        Win32ErrorCodeDescription :=
            'A communications failure occurred during a remote procedure call.';
    Win32ErrorCodes.RPC_S_UNSUPPORTED_AUTHN_LEVEL:
        Win32ErrorCodeDescription := 'The requested authentication level is not supported.';
    Win32ErrorCodes.RPC_S_NO_PRINC_NAME:
        Win32ErrorCodeDescription := 'No principal name registered.';
    Win32ErrorCodes.RPC_S_NOT_RPC_ERROR:
        Win32ErrorCodeDescription := 'The error specified is not a valid Windows RPC error code.';
    Win32ErrorCodes.RPC_S_UUID_LOCAL_ONLY:
        Win32ErrorCodeDescription :=
            'A UUID that is valid only on this computer has been allocated.';
    Win32ErrorCodes.RPC_S_SEC_PKG_ERROR:
        Win32ErrorCodeDescription := 'A security package specific error occurred.';
    Win32ErrorCodes.RPC_S_NOT_CANCELLED:
        Win32ErrorCodeDescription := 'Thread is not canceled.';
    Win32ErrorCodes.RPC_X_INVALID_ES_ACTION:
        Win32ErrorCodeDescription := 'Invalid operation on the encoding/decoding handle.';
    Win32ErrorCodes.RPC_X_WRONG_ES_VERSION:
        Win32ErrorCodeDescription := 'Incompatible version of the serializing package.';
    Win32ErrorCodes.RPC_X_WRONG_STUB_VERSION:
        Win32ErrorCodeDescription := 'Incompatible version of the RPC stub.';
    Win32ErrorCodes.RPC_X_INVALID_PIPE_OBJECT:
        Win32ErrorCodeDescription := 'The RPC pipe object is invalid or corrupted.';
    Win32ErrorCodes.RPC_X_WRONG_PIPE_ORDER:
        Win32ErrorCodeDescription := 'An invalid operation was attempted on an RPC pipe object.';
    Win32ErrorCodes.RPC_X_WRONG_PIPE_VERSION:
        Win32ErrorCodeDescription := 'Unsupported RPC pipe version.';
    Win32ErrorCodes.RPC_S_GROUP_MEMBER_NOT_FOUND:
        Win32ErrorCodeDescription := 'The group member was not found.';
    Win32ErrorCodes.EPT_S_CANT_CREATE:
        Win32ErrorCodeDescription := 'The endpoint mapper database entry could not be created.';
    Win32ErrorCodes.RPC_S_INVALID_OBJECT:
        Win32ErrorCodeDescription :=
            'The object universal unique identifier (UUID) is the nil UUID.';
    Win32ErrorCodes.ERROR_INVALID_TIME:
        Win32ErrorCodeDescription := 'The specified time is invalid.';
    Win32ErrorCodes.ERROR_INVALID_FORM_NAME:
        Win32ErrorCodeDescription := 'The specified form name is invalid.';
    Win32ErrorCodes.ERROR_INVALID_FORM_SIZE:
        Win32ErrorCodeDescription := 'The specified form size is invalid.';
    Win32ErrorCodes.ERROR_ALREADY_WAITING:
        Win32ErrorCodeDescription := 'The specified printer handle is already being waited on';
    Win32ErrorCodes.ERROR_PRINTER_DELETED:
        Win32ErrorCodeDescription := 'The specified printer has been deleted.';
    Win32ErrorCodes.ERROR_INVALID_PRINTER_STATE:
        Win32ErrorCodeDescription := 'The state of the printer is invalid.';
    Win32ErrorCodes.ERROR_PASSWORD_MUST_CHANGE:
        Win32ErrorCodeDescription :=
            'The users password must be changed before logging on the first time.';
    Win32ErrorCodes.ERROR_DOMAIN_CONTROLLER_NOT_FOUND:
        Win32ErrorCodeDescription := 'Could not find the domain controller for this domain.';
    Win32ErrorCodes.ERROR_ACCOUNT_LOCKED_OUT:
        Win32ErrorCodeDescription :=
            'The referenced account is currently locked out and may not be logged on to.';
    Win32ErrorCodes.OR_INVALID_OXID:
        Win32ErrorCodeDescription := 'The object exporter specified was not found.';
    Win32ErrorCodes.OR_INVALID_OID:
        Win32ErrorCodeDescription := 'The object specified was not found.';
    Win32ErrorCodes.OR_INVALID_SET:
        Win32ErrorCodeDescription := 'The object resolver set specified was not found.';
    Win32ErrorCodes.RPC_S_SEND_INCOMPLETE:
        Win32ErrorCodeDescription := 'Some data remains to be sent in the request buffer.';
    Win32ErrorCodes.RPC_S_INVALID_ASYNC_HANDLE:
        Win32ErrorCodeDescription := 'Invalid asynchronous remote procedure call handle.';
    Win32ErrorCodes.RPC_S_INVALID_ASYNC_CALL:
        Win32ErrorCodeDescription := 'Invalid asynchronous RPC call handle for this operation.';
    Win32ErrorCodes.RPC_X_PIPE_CLOSED:
        Win32ErrorCodeDescription := 'The RPC pipe object has already been closed.';
    Win32ErrorCodes.RPC_X_PIPE_DISCIPLINE_ERROR:
        Win32ErrorCodeDescription := 'The RPC call completed before all pipes were processed.';
    Win32ErrorCodes.RPC_X_PIPE_EMPTY:
        Win32ErrorCodeDescription := 'No more data is available from the RPC pipe.';
    Win32ErrorCodes.ERROR_NO_SITENAME:
        Win32ErrorCodeDescription := 'No site name is available for this machine.';
    Win32ErrorCodes.ERROR_CANT_ACCESS_FILE:
        Win32ErrorCodeDescription := 'The file can not be accessed by the system.';
    Win32ErrorCodes.ERROR_CANT_RESOLVE_FILENAME:
        Win32ErrorCodeDescription := 'The name of the file cannot be resolved by the system.';
    Win32ErrorCodes.RPC_S_ENTRY_TYPE_MISMATCH:
        Win32ErrorCodeDescription := 'The entry is not of the expected type.';
    Win32ErrorCodes.RPC_S_NOT_ALL_OBJS_EXPORTED:
        Win32ErrorCodeDescription :=
            'Not all object UUIDs could be exported to the specified entry.';
    Win32ErrorCodes.RPC_S_INTERFACE_NOT_EXPORTED:
        Win32ErrorCodeDescription := 'Interface could not be exported to the specified entry.';
    Win32ErrorCodes.RPC_S_PROFILE_NOT_ADDED:
        Win32ErrorCodeDescription := 'The specified profile entry could not be added.';
    Win32ErrorCodes.RPC_S_PRF_ELT_NOT_ADDED:
        Win32ErrorCodeDescription := 'The specified profile element could not be added.';
    Win32ErrorCodes.RPC_S_PRF_ELT_NOT_REMOVED:
        Win32ErrorCodeDescription := 'The specified profile element could not be removed.';
    Win32ErrorCodes.RPC_S_GRP_ELT_NOT_ADDED:
        Win32ErrorCodeDescription := 'The group element could not be added.';
    Win32ErrorCodes.RPC_S_GRP_ELT_NOT_REMOVED:
        Win32ErrorCodeDescription := 'The group element could not be removed.';
    Win32ErrorCodes.ERROR_KM_DRIVER_BLOCKED:
        Win32ErrorCodeDescription := 'The printer driver is not compatible with a policy enabled on your computer that blocks NT 4.0 drivers.';
    Win32ErrorCodes.ERROR_INVALID_PIXEL_FORMAT:
        Win32ErrorCodeDescription := 'The pixel format is invalid.';
    Win32ErrorCodes.ERROR_BAD_DRIVER:
        Win32ErrorCodeDescription := 'The specified driver is invalid.';
    Win32ErrorCodes.ERROR_INVALID_WINDOW_STYLE:
        Win32ErrorCodeDescription :=
            'The window style or class attribute is invalid for this operation.';
    Win32ErrorCodes.ERROR_METAFILE_NOT_SUPPORTED:
        Win32ErrorCodeDescription := 'The requested metafile operation is not supported.';
    Win32ErrorCodes.ERROR_TRANSFORM_NOT_SUPPORTED:
        Win32ErrorCodeDescription := 'The requested transformation operation is not supported.';
    Win32ErrorCodes.ERROR_CLIPPING_NOT_SUPPORTED:
        Win32ErrorCodeDescription := 'The requested clipping operation is not supported.';
    Win32ErrorCodes.ERROR_INVALID_CMM:
        Win32ErrorCodeDescription := 'The specified color management module is invalid.';
    Win32ErrorCodes.ERROR_INVALID_PROFILE:
        Win32ErrorCodeDescription := 'The specified color profile is invalid.';
    Win32ErrorCodes.ERROR_TAG_NOT_FOUND:
        Win32ErrorCodeDescription := 'The specified tag was not found.';
    Win32ErrorCodes.ERROR_TAG_NOT_PRESENT:
        Win32ErrorCodeDescription := 'A required tag is not present.';
    Win32ErrorCodes.ERROR_DUPLICATE_TAG:
        Win32ErrorCodeDescription := 'The specified tag is already present.';
    Win32ErrorCodes.ERROR_PROFILE_NOT_ASSOCIATED_WITH_DEVICE:
        Win32ErrorCodeDescription :=
            'The specified color profile is not associated with any device.';
    Win32ErrorCodes.ERROR_PROFILE_NOT_FOUND:
        Win32ErrorCodeDescription := 'The specified color profile was not found.';
    Win32ErrorCodes.ERROR_INVALID_COLORSPACE:
        Win32ErrorCodeDescription := 'The specified color space is invalid.';
    Win32ErrorCodes.ERROR_ICM_NOT_ENABLED:
        Win32ErrorCodeDescription := 'Image Color Management is not enabled.';
    Win32ErrorCodes.ERROR_DELETING_ICM_XFORM:
        Win32ErrorCodeDescription := 'There was an error while deleting the color transform.';
    Win32ErrorCodes.ERROR_INVALID_TRANSFORM:
        Win32ErrorCodeDescription := 'The specified color transform is invalid.';
    Win32ErrorCodes.ERROR_COLORSPACE_MISMATCH:
        Win32ErrorCodeDescription :=
            'The specified transform does not match the bitmaps color space.';
    Win32ErrorCodes.ERROR_INVALID_COLORINDEX:
        Win32ErrorCodeDescription :=
            'The specified named color index is not present in the profile.';
    Win32ErrorCodes.ERROR_CONNECTED_OTHER_PASSWORD:
        Win32ErrorCodeDescription := 'The network connection was made successfully, but the user had to be prompted for a password other than the one originally specified.';
    Win32ErrorCodes.ERROR_BAD_USERNAME:
        Win32ErrorCodeDescription := 'The specified username is invalid.';
    Win32ErrorCodes.ERROR_NOT_CONNECTED:
        Win32ErrorCodeDescription := 'This network connection does not exist.';
    Win32ErrorCodes.ERROR_OPEN_FILES:
        Win32ErrorCodeDescription := 'This network connection has files open or requests pending.';
    Win32ErrorCodes.ERROR_ACTIVE_CONNECTIONS:
        Win32ErrorCodeDescription := 'Active connections still exist.';
    Win32ErrorCodes.ERROR_DEVICE_IN_USE:
        Win32ErrorCodeDescription :=
            'The device is in use by an active process and cannot be disconnected.';
    Win32ErrorCodes.ERROR_PKINIT_FAILURE:
        Win32ErrorCodeDescription := 'The kerberos protocol encountered an error while validating the KDC certificate during smartcard logon.';
    Win32ErrorCodes.ERROR_SMARTCARD_SUBSYSTEM_FAILURE:
        Win32ErrorCodeDescription := 'The kerberos protocol encountered an error while attempting to utilize the smartcard subsystem.';
    Win32ErrorCodes.ERROR_UNKNOWN_PRINT_MONITOR:
        Win32ErrorCodeDescription := 'The specified print monitor is unknown.';
    Win32ErrorCodes.ERROR_PRINTER_DRIVER_IN_USE:
        Win32ErrorCodeDescription := 'The specified printer driver is currently in use.';
    Win32ErrorCodes.ERROR_SPOOL_FILE_NOT_FOUND:
        Win32ErrorCodeDescription := 'The spool file was not found.';
    Win32ErrorCodes.ERROR_SPL_NO_STARTDOC:
        Win32ErrorCodeDescription := 'A StartDocPrinter call was not issued.';
    Win32ErrorCodes.ERROR_SPL_NO_ADDJOB:
        Win32ErrorCodeDescription := 'An AddJob call was not issued.';
    Win32ErrorCodes.ERROR_PRINT_PROCESSOR_ALREADY_INSTALLED:
        Win32ErrorCodeDescription := 'The specified print processor has already been installed.';
    Win32ErrorCodes.ERROR_PRINT_MONITOR_ALREADY_INSTALLED:
        Win32ErrorCodeDescription := 'The specified print monitor has already been installed.';
    Win32ErrorCodes.ERROR_INVALID_PRINT_MONITOR:
        Win32ErrorCodeDescription :=
            'The specified print monitor does not have the required functions.';
    Win32ErrorCodes.ERROR_PRINT_MONITOR_IN_USE:
        Win32ErrorCodeDescription := 'The specified print monitor is currently in use.';
    Win32ErrorCodes.ERROR_PRINTER_HAS_JOBS_QUEUED:
        Win32ErrorCodeDescription :=
            'The requested operation is not allowed when there are jobs queued to the printer.';
    Win32ErrorCodes.ERROR_SUCCESS_REBOOT_REQUIRED:
        Win32ErrorCodeDescription := 'The requested operation is successful. Changes will not be effective until the system is rebooted.';
    Win32ErrorCodes.ERROR_SUCCESS_RESTART_REQUIRED:
        Win32ErrorCodeDescription := 'The requested operation is successful. Changes will not be effective until the service is restarted.';
    Win32ErrorCodes.ERROR_PRINTER_NOT_FOUND:
        Win32ErrorCodeDescription := 'No printers were found.';
    Win32ErrorCodes.ERROR_WINS_INTERNAL:
        Win32ErrorCodeDescription := 'WINS encountered an error while processing the command.';
    Win32ErrorCodes.ERROR_CAN_NOT_DEL_LOCAL_WINS:
        Win32ErrorCodeDescription := 'The local WINS can not be deleted.';
    Win32ErrorCodes.ERROR_STATIC_INIT:
        Win32ErrorCodeDescription := 'The importation from the file failed.';
    Win32ErrorCodes.ERROR_INC_BACKUP:
        Win32ErrorCodeDescription := 'The backup failed. Was a full backup done before?';
    Win32ErrorCodes.ERROR_FULL_BACKUP:
        Win32ErrorCodeDescription :=
            'The backup failed. Check the directory to which you are backing the database.';
    Win32ErrorCodes.ERROR_REC_NON_EXISTENT:
        Win32ErrorCodeDescription := 'The name does not exist in the WINS database.';
    Win32ErrorCodes.ERROR_RPL_NOT_ALLOWED:
        Win32ErrorCodeDescription := 'Replication with a nonconfigured partner is not allowed.';
    Win32ErrorCodes.ERROR_DHCP_ADDRESS_CONFLICT:
        Win32ErrorCodeDescription := 'The DHCP client has obtained an IP address that is already in use on the network. The local interface will be disabled until the DHCP client can obtain a new address.';
    Win32ErrorCodes.ERROR_WMI_GUID_NOT_FOUND:
        Win32ErrorCodeDescription :=
            'The GUID passed was not recognized as valid by a WMI data provider.';
    Win32ErrorCodes.ERROR_WMI_INSTANCE_NOT_FOUND:
        Win32ErrorCodeDescription :=
            'The instance name passed was not recognized as valid by a WMI data provider.';
    Win32ErrorCodes.ERROR_WMI_ITEMID_NOT_FOUND:
        Win32ErrorCodeDescription :=
            'The data item ID passed was not recognized as valid by a WMI data provider.';
    Win32ErrorCodes.ERROR_WMI_TRY_AGAIN:
        Win32ErrorCodeDescription :=
            'The WMI request could not be completed and should be retried.';
    Win32ErrorCodes.ERROR_WMI_DP_NOT_FOUND:
        Win32ErrorCodeDescription := 'The WMI data provider could not be located.';
    Win32ErrorCodes.ERROR_WMI_UNRESOLVED_INSTANCE_REF:
        Win32ErrorCodeDescription :=
            'The WMI data provider references an instance set that has not been registered.';
    Win32ErrorCodes.ERROR_WMI_ALREADY_ENABLED:
        Win32ErrorCodeDescription :=
            'The WMI data block or event notification has already been enabled.';
    Win32ErrorCodes.ERROR_WMI_GUID_DISCONNECTED:
        Win32ErrorCodeDescription := 'The WMI data block is no longer available.';
    Win32ErrorCodes.ERROR_WMI_SERVER_UNAVAILABLE:
        Win32ErrorCodeDescription := 'The WMI data service is not available.';
    Win32ErrorCodes.ERROR_WMI_DP_FAILED:
        Win32ErrorCodeDescription := 'The WMI data provider failed to carry out the request.';
    Win32ErrorCodes.ERROR_WMI_INVALID_MOF:
        Win32ErrorCodeDescription := 'The WMI MOF information is not valid.';
    Win32ErrorCodes.ERROR_WMI_INVALID_REGINFO:
        Win32ErrorCodeDescription := 'The WMI registration information is not valid.';
    Win32ErrorCodes.ERROR_WMI_ALREADY_DISABLED:
        Win32ErrorCodeDescription :=
            'The WMI data block or event notification has already been disabled.';
    Win32ErrorCodes.ERROR_WMI_READ_ONLY:
        Win32ErrorCodeDescription := 'The WMI data item or data block is read only.';
    Win32ErrorCodes.ERROR_WMI_SET_FAILURE:
        Win32ErrorCodeDescription := 'The WMI data item or data block could not be changed.';
    Win32ErrorCodes.ERROR_INVALID_MEDIA:
        Win32ErrorCodeDescription := 'The media identifier does not represent a valid medium.';
    Win32ErrorCodes.ERROR_INVALID_LIBRARY:
        Win32ErrorCodeDescription := 'The library identifier does not represent a valid library.';
    Win32ErrorCodes.ERROR_INVALID_MEDIA_POOL:
        Win32ErrorCodeDescription :=
            'The media pool identifier does not represent a valid media pool.';
    Win32ErrorCodes.ERROR_DRIVE_MEDIA_MISMATCH:
        Win32ErrorCodeDescription :=
            'The drive and medium are not compatible or exist in different libraries.';
    Win32ErrorCodes.ERROR_MEDIA_OFFLINE:
        Win32ErrorCodeDescription := 'The medium currently exists in an offline library and must be online to perform this operation.';
    Win32ErrorCodes.ERROR_LIBRARY_OFFLINE:
        Win32ErrorCodeDescription := 'The operation cannot be performed on an offline library.';
    Win32ErrorCodes.ERROR_EMPTY:
        Win32ErrorCodeDescription := 'The library, drive, or media pool is empty.';
    Win32ErrorCodes.ERROR_NOT_EMPTY:
        Win32ErrorCodeDescription :=
            'The library, drive, or media pool must be empty to perform this operation.';
    Win32ErrorCodes.ERROR_MEDIA_UNAVAILABLE:
        Win32ErrorCodeDescription :=
            'No media is currently available in this media pool or library.';
    Win32ErrorCodes.ERROR_RESOURCE_DISABLED:
        Win32ErrorCodeDescription := 'A resource required for this operation is disabled.';
    Win32ErrorCodes.ERROR_INVALID_CLEANER:
        Win32ErrorCodeDescription := 'The media identifier does not represent a valid cleaner.';
    Win32ErrorCodes.ERROR_UNABLE_TO_CLEAN:
        Win32ErrorCodeDescription := 'The drive cannot be cleaned or does not support cleaning.';
    Win32ErrorCodes.ERROR_OBJECT_NOT_FOUND:
        Win32ErrorCodeDescription := 'The object identifier does not represent a valid object.';
    Win32ErrorCodes.ERROR_DATABASE_FAILURE:
        Win32ErrorCodeDescription := 'Unable to read from or write to the database.';
    Win32ErrorCodes.ERROR_DATABASE_FULL:
        Win32ErrorCodeDescription := 'The database is full.';
    Win32ErrorCodes.ERROR_MEDIA_INCOMPATIBLE:
        Win32ErrorCodeDescription := 'The medium is not compatible with the device or media pool.';
    Win32ErrorCodes.ERROR_RESOURCE_NOT_PRESENT:
        Win32ErrorCodeDescription := 'The resource required for this operation does not exist.';
    Win32ErrorCodes.ERROR_INVALID_OPERATION:
        Win32ErrorCodeDescription := 'The operation identifier is not valid.';
    Win32ErrorCodes.ERROR_MEDIA_NOT_AVAILABLE:
        Win32ErrorCodeDescription := 'The media is not mounted or ready for use.';
    Win32ErrorCodes.ERROR_DEVICE_NOT_AVAILABLE:
        Win32ErrorCodeDescription := 'The device is not ready for use.';
    Win32ErrorCodes.ERROR_REQUEST_REFUSED:
        Win32ErrorCodeDescription := 'The operator or administrator has refused the request.';
    Win32ErrorCodes.ERROR_INVALID_DRIVE_OBJECT:
        Win32ErrorCodeDescription := 'The drive identifier does not represent a valid drive.';
    Win32ErrorCodes.ERROR_LIBRARY_FULL:
        Win32ErrorCodeDescription := 'Library is full. No slot is available for use.';
    Win32ErrorCodes.ERROR_MEDIUM_NOT_ACCESSIBLE:
        Win32ErrorCodeDescription := 'The transport cannot access the medium.';
    Win32ErrorCodes.ERROR_UNABLE_TO_LOAD_MEDIUM:
        Win32ErrorCodeDescription := 'Unable to load the medium into the drive.';
    Win32ErrorCodes.ERROR_UNABLE_TO_INVENTORY_DRIVE:
        Win32ErrorCodeDescription := 'Unable to retrieve status about the drive.';
    Win32ErrorCodes.ERROR_UNABLE_TO_INVENTORY_SLOT:
        Win32ErrorCodeDescription := 'Unable to retrieve status about the slot.';
    Win32ErrorCodes.ERROR_UNABLE_TO_INVENTORY_TRANSPORT:
        Win32ErrorCodeDescription := 'Unable to retrieve status about the transport.';
    Win32ErrorCodes.ERROR_TRANSPORT_FULL:
        Win32ErrorCodeDescription := 'Cannot use the transport because it is already in use.';
    Win32ErrorCodes.ERROR_CONTROLLING_IEPORT:
        Win32ErrorCodeDescription := 'Unable to open or close the inject/eject port.';
    Win32ErrorCodes.ERROR_UNABLE_TO_EJECT_MOUNTED_MEDIA:
        Win32ErrorCodeDescription := 'Unable to eject the media because it is in a drive.';
    Win32ErrorCodes.ERROR_CLEANER_SLOT_SET:
        Win32ErrorCodeDescription := 'A cleaner slot is already reserved.';
    Win32ErrorCodes.ERROR_CLEANER_SLOT_NOT_SET:
        Win32ErrorCodeDescription := 'A cleaner slot is not reserved.';
    Win32ErrorCodes.ERROR_CLEANER_CARTRIDGE_SPENT:
        Win32ErrorCodeDescription :=
            'The cleaner cartridge has performed the maximum number of drive cleanings.';
    Win32ErrorCodes.ERROR_UNEXPECTED_OMID:
        Win32ErrorCodeDescription := 'Unexpected on-medium identifier.';
    Win32ErrorCodes.ERROR_CANT_DELETE_LAST_ITEM:
        Win32ErrorCodeDescription :=
            'The last remaining item in this group or resource cannot be deleted.';
    Win32ErrorCodes.ERROR_MESSAGE_EXCEEDS_MAX_SIZE:
        Win32ErrorCodeDescription :=
            'The message provided exceeds the maximum size allowed for this parameter.';
    Win32ErrorCodes.ERROR_VOLUME_CONTAINS_SYS_FILES:
        Win32ErrorCodeDescription := 'The volume contains system or paging files.';
    Win32ErrorCodes.ERROR_INDIGENOUS_TYPE:
        Win32ErrorCodeDescription := 'The media type cannot be removed from this library since at least one drive in the library reports it can support this media type.';
    Win32ErrorCodes.ERROR_NO_SUPPORTING_DRIVES:
        Win32ErrorCodeDescription := 'This offline media cannot be mounted on this system since no enabled drives are present which can be used.';
    Win32ErrorCodes.ERROR_CLEANER_CARTRIDGE_INSTALLED:
        Win32ErrorCodeDescription := 'A cleaner cartridge is present in the tape library.';
    Win32ErrorCodes.ERROR_FILE_OFFLINE:
        Win32ErrorCodeDescription := 'The remote storage service was not able to recall the file.';
    Win32ErrorCodes.ERROR_REMOTE_STORAGE_NOT_ACTIVE:
        Win32ErrorCodeDescription := 'The remote storage service is not operational at this time.';
    Win32ErrorCodes.ERROR_REMOTE_STORAGE_MEDIA_ERROR:
        Win32ErrorCodeDescription := 'The remote storage service encountered a media error.';
    Win32ErrorCodes.ERROR_NOT_A_REPARSE_POINT:
        Win32ErrorCodeDescription := 'The file or directory is not a reparse point.';
    Win32ErrorCodes.ERROR_REPARSE_ATTRIBUTE_CONFLICT:
        Win32ErrorCodeDescription := 'The reparse point attribute cannot be set because it conflicts with an existing attribute.';
    Win32ErrorCodes.ERROR_INVALID_REPARSE_DATA:
        Win32ErrorCodeDescription := 'The data present in the reparse point buffer is invalid.';
    Win32ErrorCodes.ERROR_REPARSE_TAG_INVALID:
        Win32ErrorCodeDescription := 'The tag present in the reparse point buffer is invalid.';
    Win32ErrorCodes.ERROR_REPARSE_TAG_MISMATCH:
        Win32ErrorCodeDescription := 'There is a mismatch between the tag specified in the request and the tag present in the reparse point.';
    Win32ErrorCodes.ERROR_VOLUME_NOT_SIS_ENABLED:
        Win32ErrorCodeDescription := 'Single Instance Storage is not available on this volume.';
    Win32ErrorCodes.ERROR_DEPENDENT_RESOURCE_EXISTS:
        Win32ErrorCodeDescription := 'The cluster resource cannot be moved to another group because other resources are dependent on it.';
    Win32ErrorCodes.ERROR_DEPENDENCY_NOT_FOUND:
        Win32ErrorCodeDescription := 'The cluster resource dependency cannot be found.';
    Win32ErrorCodes.ERROR_DEPENDENCY_ALREADY_EXISTS:
        Win32ErrorCodeDescription := 'The cluster resource cannot be made dependent on the specified resource because it is already dependent.';
    Win32ErrorCodes.ERROR_RESOURCE_NOT_ONLINE:
        Win32ErrorCodeDescription := 'The cluster resource is not online.';
    Win32ErrorCodes.ERROR_HOST_NODE_NOT_AVAILABLE:
        Win32ErrorCodeDescription := 'A cluster node is not available for this operation.';
    Win32ErrorCodes.ERROR_RESOURCE_NOT_AVAILABLE:
        Win32ErrorCodeDescription := 'The cluster resource is not available.';
    Win32ErrorCodes.ERROR_RESOURCE_NOT_FOUND:
        Win32ErrorCodeDescription := 'The cluster resource could not be found.';
    Win32ErrorCodes.ERROR_SHUTDOWN_CLUSTER:
        Win32ErrorCodeDescription := 'The cluster is being shut down.';
    Win32ErrorCodes.ERROR_CANT_EVICT_ACTIVE_NODE:
        Win32ErrorCodeDescription :=
            'A cluster node cannot be evicted from the cluster unless the node is down.';
    Win32ErrorCodes.ERROR_OBJECT_ALREADY_EXISTS:
        Win32ErrorCodeDescription := 'The object already exists.';
    Win32ErrorCodes.ERROR_OBJECT_IN_LIST:
        Win32ErrorCodeDescription := 'The object is already in the list.';
    Win32ErrorCodes.ERROR_GROUP_NOT_AVAILABLE:
        Win32ErrorCodeDescription := 'The cluster group is not available for any new requests.';
    Win32ErrorCodes.ERROR_GROUP_NOT_FOUND:
        Win32ErrorCodeDescription := 'The cluster group could not be found.';
    Win32ErrorCodes.ERROR_GROUP_NOT_ONLINE:
        Win32ErrorCodeDescription :=
            'The operation could not be completed because the cluster group is not online.';
    Win32ErrorCodes.ERROR_HOST_NODE_NOT_RESOURCE_OWNER:
        Win32ErrorCodeDescription := 'The cluster node is not the owner of the resource.';
    Win32ErrorCodes.ERROR_HOST_NODE_NOT_GROUP_OWNER:
        Win32ErrorCodeDescription := 'The cluster node is not the owner of the group.';
    Win32ErrorCodes.ERROR_RESMON_CREATE_FAILED:
        Win32ErrorCodeDescription :=
            'The cluster resource could not be created in the specified resource monitor.';
    Win32ErrorCodes.ERROR_RESMON_ONLINE_FAILED:
        Win32ErrorCodeDescription :=
            'The cluster resource could not be brought online by the resource monitor.';
    Win32ErrorCodes.ERROR_RESOURCE_ONLINE:
        Win32ErrorCodeDescription :=
            'The operation could not be completed because the cluster resource is online.';
    Win32ErrorCodes.ERROR_QUORUM_RESOURCE:
        Win32ErrorCodeDescription := 'The cluster resource could not be deleted or brought offline because it is the quorum resource.';
    Win32ErrorCodes.ERROR_NOT_QUORUM_CAPABLE:
        Win32ErrorCodeDescription := 'The cluster could not make the specified resource a quorum resource because it is not capable of being a quorum resource.';
    Win32ErrorCodes.ERROR_CLUSTER_SHUTTING_DOWN:
        Win32ErrorCodeDescription := 'The cluster software is shutting down.';
    Win32ErrorCodes.ERROR_INVALID_STATE:
        Win32ErrorCodeDescription :=
            'The group or resource is not in the correct state to perform the requested operation.';
    Win32ErrorCodes.ERROR_RESOURCE_PROPERTIES_STORED:
        Win32ErrorCodeDescription := 'The properties were stored but not all changes will take effect until the next time the resource is brought online.';
    Win32ErrorCodes.ERROR_NOT_QUORUM_CLASS:
        Win32ErrorCodeDescription := 'The cluster could not make the specified resource a quorum resource because it does not belong to a shared storage class.';
    Win32ErrorCodes.ERROR_CORE_RESOURCE:
        Win32ErrorCodeDescription :=
            'The cluster resource could not be deleted since it is a core resource.';
    Win32ErrorCodes.ERROR_QUORUM_RESOURCE_ONLINE_FAILED:
        Win32ErrorCodeDescription := 'The quorum resource failed to come online.';
    Win32ErrorCodes.ERROR_QUORUMLOG_OPEN_FAILED:
        Win32ErrorCodeDescription :=
            'The quorum log could not be created or mounted successfully.';
    Win32ErrorCodes.ERROR_CLUSTERLOG_CORRUPT:
        Win32ErrorCodeDescription := 'The cluster log is corrupt.';
    Win32ErrorCodes.ERROR_CLUSTERLOG_RECORD_EXCEEDS_MAXSIZE:
        Win32ErrorCodeDescription :=
            'The record could not be written to the cluster log since it exceeds the maximum size.';
    Win32ErrorCodes.ERROR_CLUSTERLOG_EXCEEDS_MAXSIZE:
        Win32ErrorCodeDescription := 'The cluster log exceeds its maximum size.';
    Win32ErrorCodes.ERROR_CLUSTERLOG_CHKPOINT_NOT_FOUND:
        Win32ErrorCodeDescription := 'No checkpoint record was found in the cluster log.';
    Win32ErrorCodes.ERROR_CLUSTERLOG_NOT_ENOUGH_SPACE:
        Win32ErrorCodeDescription :=
            'The minimum required disk space needed for logging is not available.';
    Win32ErrorCodes.ERROR_QUORUM_OWNER_ALIVE:
        Win32ErrorCodeDescription := 'The cluster node failed to take control of the quorum resource because the resource is owned by another active node.';
    Win32ErrorCodes.ERROR_NETWORK_NOT_AVAILABLE:
        Win32ErrorCodeDescription := 'A cluster network is not available for this operation.';
    Win32ErrorCodes.ERROR_NODE_NOT_AVAILABLE:
        Win32ErrorCodeDescription := 'A cluster node is not available for this operation.';
    Win32ErrorCodes.ERROR_ALL_NODES_NOT_AVAILABLE:
        Win32ErrorCodeDescription :=
            'All cluster nodes must be running to perform this operation.';
    Win32ErrorCodes.ERROR_RESOURCE_FAILED:
        Win32ErrorCodeDescription := 'A cluster resource failed.';
    Win32ErrorCodes.ERROR_CLUSTER_INVALID_NODE:
        Win32ErrorCodeDescription := 'The cluster node is not valid.';
    Win32ErrorCodes.ERROR_CLUSTER_NODE_EXISTS:
        Win32ErrorCodeDescription := 'The cluster node already exists.';
    Win32ErrorCodes.ERROR_CLUSTER_JOIN_IN_PROGRESS:
        Win32ErrorCodeDescription := 'A node is in the process of joining the cluster.';
    Win32ErrorCodes.ERROR_CLUSTER_NODE_NOT_FOUND:
        Win32ErrorCodeDescription := 'The cluster node was not found.';
    Win32ErrorCodes.ERROR_CLUSTER_LOCAL_NODE_NOT_FOUND:
        Win32ErrorCodeDescription := 'The cluster local node information was not found.';
    Win32ErrorCodes.ERROR_CLUSTER_NETWORK_EXISTS:
        Win32ErrorCodeDescription := 'The cluster network already exists.';
    Win32ErrorCodes.ERROR_CLUSTER_NETWORK_NOT_FOUND:
        Win32ErrorCodeDescription := 'The cluster network was not found.';
    Win32ErrorCodes.ERROR_CLUSTER_NETINTERFACE_EXISTS:
        Win32ErrorCodeDescription := 'The cluster network interface already exists.';
    Win32ErrorCodes.ERROR_CLUSTER_NETINTERFACE_NOT_FOUND:
        Win32ErrorCodeDescription := 'The cluster network interface was not found.';
    Win32ErrorCodes.ERROR_CLUSTER_INVALID_REQUEST:
        Win32ErrorCodeDescription := 'The cluster request is not valid for this object.';
    Win32ErrorCodes.ERROR_CLUSTER_INVALID_NETWORK_PROVIDER:
        Win32ErrorCodeDescription := 'The cluster network provider is not valid.';
    Win32ErrorCodes.ERROR_CLUSTER_NODE_DOWN:
        Win32ErrorCodeDescription := 'The cluster node is down.';
    Win32ErrorCodes.ERROR_CLUSTER_NODE_UNREACHABLE:
        Win32ErrorCodeDescription := 'The cluster node is not reachable.';
    Win32ErrorCodes.ERROR_CLUSTER_NODE_NOT_MEMBER:
        Win32ErrorCodeDescription := 'The cluster node is not a member of the cluster.';
    Win32ErrorCodes.ERROR_CLUSTER_JOIN_NOT_IN_PROGRESS:
        Win32ErrorCodeDescription := 'A cluster join operation is not in progress.';
    Win32ErrorCodes.ERROR_CLUSTER_INVALID_NETWORK:
        Win32ErrorCodeDescription := 'The cluster network is not valid.';
    Win32ErrorCodes.ERROR_CLUSTER_NODE_UP:
        Win32ErrorCodeDescription := 'The cluster node is up.';
    Win32ErrorCodes.ERROR_CLUSTER_IPADDR_IN_USE:
        Win32ErrorCodeDescription := 'The cluster IP address is already in use.';
    Win32ErrorCodes.ERROR_CLUSTER_NODE_NOT_PAUSED:
        Win32ErrorCodeDescription := 'The cluster node is not paused.';
    Win32ErrorCodes.ERROR_CLUSTER_NO_SECURITY_CONTEXT:
        Win32ErrorCodeDescription := 'No cluster security context is available.';
    Win32ErrorCodes.ERROR_CLUSTER_NETWORK_NOT_INTERNAL:
        Win32ErrorCodeDescription :=
            'The cluster network is not configured for internal cluster communication.';
    Win32ErrorCodes.ERROR_CLUSTER_NODE_ALREADY_UP:
        Win32ErrorCodeDescription := 'The cluster node is already up.';
    Win32ErrorCodes.ERROR_CLUSTER_NODE_ALREADY_DOWN:
        Win32ErrorCodeDescription := 'The cluster node is already down.';
    Win32ErrorCodes.ERROR_CLUSTER_NETWORK_ALREADY_ONLINE:
        Win32ErrorCodeDescription := 'The cluster network is already online.';
    Win32ErrorCodes.ERROR_CLUSTER_NETWORK_ALREADY_OFFLINE:
        Win32ErrorCodeDescription := 'The cluster network is already offline.';
    Win32ErrorCodes.ERROR_CLUSTER_NODE_ALREADY_MEMBER:
        Win32ErrorCodeDescription := 'The cluster node is already a member of the cluster.';
    Win32ErrorCodes.ERROR_CLUSTER_LAST_INTERNAL_NETWORK:
        Win32ErrorCodeDescription := 'The cluster network is the only one configured for internal cluster communication between two or more active cluster nodes. The internal communication capability cannot be removed from the network.';
    Win32ErrorCodes.ERROR_CLUSTER_NETWORK_HAS_DEPENDENTS:
        Win32ErrorCodeDescription := 'One or more cluster resources depend on the network to provide service to clients. The client access capability cannot be removed from the network.';
    Win32ErrorCodes.ERROR_INVALID_OPERATION_ON_QUORUM:
        Win32ErrorCodeDescription := 'This operation cannot be performed on the cluster resource as it the quorum resource. You may not bring the quorum resource offline or modify its possible owners list.';
    Win32ErrorCodes.ERROR_DEPENDENCY_NOT_ALLOWED:
        Win32ErrorCodeDescription :=
            'The cluster quorum resource is not allowed to have any dependencies.';
    Win32ErrorCodes.ERROR_CLUSTER_NODE_PAUSED:
        Win32ErrorCodeDescription := 'The cluster node is paused.';
    Win32ErrorCodes.ERROR_NODE_CANT_HOST_RESOURCE:
        Win32ErrorCodeDescription :=
            'The cluster resource cannot be brought online. The owner node cannot run this resource.';
    Win32ErrorCodes.ERROR_CLUSTER_NODE_NOT_READY:
        Win32ErrorCodeDescription :=
            'The cluster node is not ready to perform the requested operation.';
    Win32ErrorCodes.ERROR_CLUSTER_NODE_SHUTTING_DOWN:
        Win32ErrorCodeDescription := 'The cluster node is shutting down.';
    Win32ErrorCodes.ERROR_CLUSTER_JOIN_ABORTED:
        Win32ErrorCodeDescription := 'The cluster join operation was aborted.';
    Win32ErrorCodes.ERROR_CLUSTER_INCOMPATIBLE_VERSIONS:
        Win32ErrorCodeDescription := 'The cluster join operation failed due to incompatible software versions between the joining node and its sponsor.';
    Win32ErrorCodes.ERROR_CLUSTER_MAXNUM_OF_RESOURCES_EXCEEDED:
        Win32ErrorCodeDescription := 'This resource cannot be created because the cluster has reached the limit on the number of resources it can monitor.';
    Win32ErrorCodes.ERROR_CLUSTER_SYSTEM_CONFIG_CHANGED:
        Win32ErrorCodeDescription := 'The system configuration changed during the cluster join or form operation. The join or form operation was aborted.';
    Win32ErrorCodes.ERROR_CLUSTER_RESOURCE_TYPE_NOT_FOUND:
        Win32ErrorCodeDescription := 'The specified resource type was not found.';
    Win32ErrorCodes.ERROR_CLUSTER_RESTYPE_NOT_SUPPORTED:
        Win32ErrorCodeDescription := 'The specified node does not support a resource of this type. This may be due to version inconsistencies or due to the absence of the resource DLL on this node.';
    Win32ErrorCodes.ERROR_CLUSTER_RESNAME_NOT_FOUND:
        Win32ErrorCodeDescription := 'The specified resource name is supported by this resource DLL. This may be due to a bad (or changed) name supplied to the resource DLL.';
    Win32ErrorCodes.ERROR_CLUSTER_NO_RPC_PACKAGES_REGISTERED:
        Win32ErrorCodeDescription :=
            'No authentication package could be registered with the RPC server.';
    Win32ErrorCodes.ERROR_CLUSTER_OWNER_NOT_IN_PREFLIST:
        Win32ErrorCodeDescription := 'You cannot bring the group online because the owner of the group is not in the preferred list for the group. To change the owner node for the group, move the group.';
    Win32ErrorCodes.ERROR_CLUSTER_DATABASE_SEQMISMATCH:
        Win32ErrorCodeDescription := 'The join operation failed because the cluster database sequence number has changed or is incompatible with the locker node. This may happen during a join operation if the cluster database was changing during the join.';
    Win32ErrorCodes.ERROR_RESMON_INVALID_STATE:
        Win32ErrorCodeDescription := 'The resource monitor will not allow the fail operation to be performed while the resource is in its current state. This may happen if the resource is in a pending state.';
    Win32ErrorCodes.ERROR_CLUSTER_GUM_NOT_LOCKER:
        Win32ErrorCodeDescription :=
            'A non locker code got a request to reserve the lock for making global updates.';
    Win32ErrorCodes.ERROR_QUORUM_DISK_NOT_FOUND:
        Win32ErrorCodeDescription :=
            'The quorum disk could not be located by the cluster service.';
    Win32ErrorCodes.ERROR_DATABASE_BACKUP_CORRUPT:
        Win32ErrorCodeDescription := 'The backup up cluster database is possibly corrupt.';
    Win32ErrorCodes.ERROR_CLUSTER_NODE_ALREADY_HAS_DFS_ROOT:
        Win32ErrorCodeDescription := 'A DFS root already exists in this cluster node.';
    Win32ErrorCodes.ERROR_RESOURCE_PROPERTY_UNCHANGEABLE:
        Win32ErrorCodeDescription := 'An attempt to modify a resource property failed because it conflicts with another existing property.';
    Win32ErrorCodes.ERROR_CLUSTER_MEMBERSHIP_INVALID_STATE:
        Win32ErrorCodeDescription := 'An operation was attempted that is incompatible with the current membership state of the node.';
    Win32ErrorCodes.ERROR_CLUSTER_QUORUMLOG_NOT_FOUND:
        Win32ErrorCodeDescription := 'The quorum resource does not contain the quorum log.';
    Win32ErrorCodes.ERROR_CLUSTER_MEMBERSHIP_HALT:
        Win32ErrorCodeDescription :=
            'The membership engine requested shutdown of the cluster service on this node.';
    Win32ErrorCodes.ERROR_CLUSTER_INSTANCE_ID_MISMATCH:
        Win32ErrorCodeDescription := 'The join operation failed because the cluster instance ID of the joining node does not match the cluster instance ID of the sponsor node.';
    Win32ErrorCodes.ERROR_CLUSTER_NETWORK_NOT_FOUND_FOR_IP:
        Win32ErrorCodeDescription := 'A matching network for the specified IP address could not be found. Please also specify a subnet mask and a cluster network.';
    Win32ErrorCodes.ERROR_CLUSTER_PROPERTY_DATA_TYPE_MISMATCH:
        Win32ErrorCodeDescription := 'The actual data type of the property did not match the expected data type of the property.';
    Win32ErrorCodes.ERROR_CLUSTER_EVICT_WITHOUT_CLEANUP:
        Win32ErrorCodeDescription := 'The cluster node was evicted from the cluster successfully. The node was not cleaned up because it does not support the evict cleanup functionality.';
    Win32ErrorCodes.ERROR_ENCRYPTION_FAILED:
        Win32ErrorCodeDescription := 'The specified file could not be encrypted.';
    Win32ErrorCodes.ERROR_DECRYPTION_FAILED:
        Win32ErrorCodeDescription := 'The specified file could not be decrypted.';
    Win32ErrorCodes.ERROR_FILE_ENCRYPTED:
        Win32ErrorCodeDescription :=
            'The specified file is encrypted and the user does not have the ability to decrypt it.';
    Win32ErrorCodes.ERROR_NO_RECOVERY_POLICY:
        Win32ErrorCodeDescription :=
            'There is no valid encryption recovery policy configured for this system.';
    Win32ErrorCodes.ERROR_NO_EFS:
        Win32ErrorCodeDescription :=
            'The required encryption driver is not loaded for this system.';
    Win32ErrorCodes.ERROR_WRONG_EFS:
        Win32ErrorCodeDescription :=
            'The file was encrypted with a different encryption driver than is currently loaded.';
    Win32ErrorCodes.ERROR_NO_USER_KEYS:
        Win32ErrorCodeDescription := 'There are no EFS keys defined for the user.';
    Win32ErrorCodes.ERROR_FILE_NOT_ENCRYPTED:
        Win32ErrorCodeDescription := 'The specified file is not encrypted.';
    Win32ErrorCodes.ERROR_NOT_EXPORT_FORMAT:
        Win32ErrorCodeDescription := 'The specified file is not in the defined EFS export format.';
    Win32ErrorCodes.ERROR_FILE_READ_ONLY:
        Win32ErrorCodeDescription := 'The specified file is read only.';
    Win32ErrorCodes.ERROR_DIR_EFS_DISALLOWED:
        Win32ErrorCodeDescription := 'The directory has been disabled for encryption.';
    Win32ErrorCodes.ERROR_EFS_SERVER_NOT_TRUSTED:
        Win32ErrorCodeDescription := 'The server is not trusted for remote encryption operation.';
    Win32ErrorCodes.ERROR_BAD_RECOVERY_POLICY:
        Win32ErrorCodeDescription :=
            'Recovery policy configured for this system contains invalid recovery certificate.';
    Win32ErrorCodes.ERROR_EFS_ALG_BLOB_TOO_BIG:
        Win32ErrorCodeDescription := 'The encryption algorithm used on the source file needs a bigger key buffer than the one on the destination file.';
    Win32ErrorCodes.ERROR_VOLUME_NOT_SUPPORT_EFS:
        Win32ErrorCodeDescription := 'The disk partition does not support file encryption.';
    Win32ErrorCodes.ERROR_NO_BROWSER_SERVERS_FOUND:
        Win32ErrorCodeDescription :=
            'The list of servers for this workgroup is not currently available.';
    Win32ErrorCodes.SCHED_E_SERVICE_NOT_LOCALSYSTEM:
        Win32ErrorCodeDescription := 'The Task Scheduler service must be configured to run in the System account to function properly. Individual tasks may be configured to run in other accounts.';
    Win32ErrorCodes.ERROR_CTX_WINSTATION_NAME_INVALID:
        Win32ErrorCodeDescription := 'The specified session name is invalid.';
    Win32ErrorCodes.ERROR_CTX_INVALID_PD:
        Win32ErrorCodeDescription := 'The specified protocol driver is invalid.';
    Win32ErrorCodes.ERROR_CTX_PD_NOT_FOUND:
        Win32ErrorCodeDescription :=
            'The specified protocol driver was not found in the system path.';
    Win32ErrorCodes.ERROR_CTX_WD_NOT_FOUND:
        Win32ErrorCodeDescription :=
            'The specified terminal connection driver was not found in the system path.';
    Win32ErrorCodes.ERROR_CTX_CANNOT_MAKE_EVENTLOG_ENTRY:
        Win32ErrorCodeDescription :=
            'A registry key for event logging could not be created for this session.';
    Win32ErrorCodes.ERROR_CTX_SERVICE_NAME_COLLISION:
        Win32ErrorCodeDescription := 'A service with the same name already exists on the system.';
    Win32ErrorCodes.ERROR_CTX_CLOSE_PENDING:
        Win32ErrorCodeDescription := 'A close operation is pending on the session.';
    Win32ErrorCodes.ERROR_CTX_NO_OUTBUF:
        Win32ErrorCodeDescription := 'There are no free output buffers available.';
    Win32ErrorCodes.ERROR_CTX_MODEM_INF_NOT_FOUND:
        Win32ErrorCodeDescription := 'The MODEM.INF file was not found.';
    Win32ErrorCodes.ERROR_CTX_INVALID_MODEMNAME:
        Win32ErrorCodeDescription := 'The modem name was not found in MODEM.INF.';
    Win32ErrorCodes.ERROR_CTX_MODEM_RESPONSE_ERROR:
        Win32ErrorCodeDescription := 'The modem did not accept the command sent to it. Verify that the configured modem name matches the attached modem.';
    Win32ErrorCodes.ERROR_CTX_MODEM_RESPONSE_TIMEOUT:
        Win32ErrorCodeDescription := 'The modem did not respond to the command sent to it. Verify that the modem is properly cabled and powered on.';
    Win32ErrorCodes.ERROR_CTX_MODEM_RESPONSE_NO_CARRIER:
        Win32ErrorCodeDescription :=
            'Carrier detect has failed or carrier has been dropped due to disconnect.';
    Win32ErrorCodes.ERROR_CTX_MODEM_RESPONSE_NO_DIALTONE:
        Win32ErrorCodeDescription := 'Dial tone not detected within the required time. Verify that the phone cable is properly attached and functional.';
    Win32ErrorCodes.ERROR_CTX_MODEM_RESPONSE_BUSY:
        Win32ErrorCodeDescription := 'Busy signal detected at remote site on callback.';
    Win32ErrorCodes.ERROR_CTX_MODEM_RESPONSE_VOICE:
        Win32ErrorCodeDescription := 'Voice detected at remote site on callback.';
    Win32ErrorCodes.ERROR_CTX_TD_ERROR:
        Win32ErrorCodeDescription := 'Transport driver error';
    Win32ErrorCodes.ERROR_CTX_WINSTATION_NOT_FOUND:
        Win32ErrorCodeDescription := 'The specified session cannot be found.';
    Win32ErrorCodes.ERROR_CTX_WINSTATION_ALREADY_EXISTS:
        Win32ErrorCodeDescription := 'The specified session name is already in use.';
    Win32ErrorCodes.ERROR_CTX_WINSTATION_BUSY:
        Win32ErrorCodeDescription := 'The requested operation cannot be completed because the terminal connection is currently busy processing a connect, disconnect, reset, or delete operation.';
    Win32ErrorCodes.ERROR_CTX_BAD_VIDEO_MODE:
        Win32ErrorCodeDescription := 'An attempt has been made to connect to a session whose video mode is not supported by the current client.';
    Win32ErrorCodes.ERROR_CTX_GRAPHICS_INVALID:
        Win32ErrorCodeDescription := 'The application attempted to enable DOS graphics mode. DOS graphics mode is not supported.';
    Win32ErrorCodes.ERROR_CTX_LOGON_DISABLED:
        Win32ErrorCodeDescription :=
            'Your interactive logon privilege has been disabled. Please contact your administrator.';
    Win32ErrorCodes.ERROR_CTX_NOT_CONSOLE:
        Win32ErrorCodeDescription := 'The requested operation can be performed only on the system console. This is most often the result of a driver or system DLL requiring direct console access.';
    Win32ErrorCodes.ERROR_CTX_CLIENT_QUERY_TIMEOUT:
        Win32ErrorCodeDescription := 'The client failed to respond to the server connect message.';
    Win32ErrorCodes.ERROR_CTX_CONSOLE_DISCONNECT:
        Win32ErrorCodeDescription := 'Disconnecting the console session is not supported.';
    Win32ErrorCodes.ERROR_CTX_CONSOLE_CONNECT:
        Win32ErrorCodeDescription :=
            'Reconnecting a disconnected session to the console is not supported.';
    Win32ErrorCodes.ERROR_CTX_SHADOW_DENIED:
        Win32ErrorCodeDescription := 'The request to control another session remotely was denied.';
    Win32ErrorCodes.ERROR_CTX_WINSTATION_ACCESS_DENIED:
        Win32ErrorCodeDescription := 'The requested session access is denied.';
    Win32ErrorCodes.ERROR_CTX_INVALID_WD:
        Win32ErrorCodeDescription := 'The specified terminal connection driver is invalid.';
    Win32ErrorCodes.ERROR_CTX_SHADOW_INVALID:
        Win32ErrorCodeDescription := 'The requested session cannot be controlled remotely. This may be because the session is disconnected or does not currently have a user logged on.';
    Win32ErrorCodes.ERROR_CTX_SHADOW_DISABLED:
        Win32ErrorCodeDescription :=
            'The requested session is not configured to allow remote control.';
    Win32ErrorCodes.ERROR_CTX_CLIENT_LICENSE_IN_USE:
        Win32ErrorCodeDescription := 'Your request to connect to this Terminal Server has been rejected. Your Terminal Server client license number is currently being used by another user. Please call your system administrator to obtain a unique license number.';
    Win32ErrorCodes.ERROR_CTX_CLIENT_LICENSE_NOT_SET:
        Win32ErrorCodeDescription := 'Your request to connect to this Terminal Server has been rejected. Your Terminal Server client license number has not been entered for this copy of the Terminal Server client. Please contact your system administrator.';
    Win32ErrorCodes.ERROR_CTX_LICENSE_NOT_AVAILABLE:
        Win32ErrorCodeDescription :=
            'The system has reached its licensed logon limit. Please try again later.';
    Win32ErrorCodes.ERROR_CTX_LICENSE_CLIENT_INVALID:
        Win32ErrorCodeDescription := 'The client you are using is not licensed to use this system. Your logon request is denied.';
    Win32ErrorCodes.ERROR_CTX_LICENSE_EXPIRED:
        Win32ErrorCodeDescription :=
            'The system license has expired. Your logon request is denied.';
    Win32ErrorCodes.ERROR_CTX_SHADOW_NOT_RUNNING:
        Win32ErrorCodeDescription := 'Remote control could not be terminated because the specified session is not currently being remotely controlled.';
    Win32ErrorCodes.FRS_ERR_INVALID_API_SEQUENCE:
        Win32ErrorCodeDescription := 'The file replication service API was called incorrectly.';
    Win32ErrorCodes.FRS_ERR_STARTING_SERVICE:
        Win32ErrorCodeDescription := 'The file replication service cannot be started.';
    Win32ErrorCodes.FRS_ERR_STOPPING_SERVICE:
        Win32ErrorCodeDescription := 'The file replication service cannot be stopped.';
    Win32ErrorCodes.FRS_ERR_INTERNAL_API:
        Win32ErrorCodeDescription := 'The file replication service API terminated the request. The event log may have more information.';
    Win32ErrorCodes.FRS_ERR_INTERNAL:
        Win32ErrorCodeDescription := 'The file replication service terminated the request. The event log may have more information.';
    Win32ErrorCodes.FRS_ERR_SERVICE_COMM:
        Win32ErrorCodeDescription := 'The file replication service cannot be contacted. The event log may have more information.';
    Win32ErrorCodes.FRS_ERR_INSUFFICIENT_PRIV:
        Win32ErrorCodeDescription := 'The file replication service cannot satisfy the request because the user has insufficient privileges. The event log may have more information.';
    Win32ErrorCodes.FRS_ERR_AUTHENTICATION:
        Win32ErrorCodeDescription := 'The file replication service cannot satisfy the request because authenticated RPC is not available. The event log may have more information.';
    Win32ErrorCodes.FRS_ERR_PARENT_INSUFFICIENT_PRIV:
        Win32ErrorCodeDescription := 'The file replication service cannot satisfy the request because the user has insufficient privileges on the domain controller. The event log may have more information.';
    Win32ErrorCodes.FRS_ERR_PARENT_AUTHENTICATION:
        Win32ErrorCodeDescription := 'The file replication service cannot satisfy the request because authenticated RPC is not available on the domain controller. The event log may have more information.';
    Win32ErrorCodes.FRS_ERR_CHILD_TO_PARENT_COMM:
        Win32ErrorCodeDescription := 'The file replication service cannot communicate with the file replication service on the domain controller. The event log may have more information.';
    Win32ErrorCodes.FRS_ERR_PARENT_TO_CHILD_COMM:
        Win32ErrorCodeDescription := 'The file replication service on the domain controller cannot communicate with the file replication service on this computer. The event log may have more information.';
    Win32ErrorCodes.FRS_ERR_SYSVOL_POPULATE:
        Win32ErrorCodeDescription := 'The file replication service cannot populate the system volume because of an internal error. The event log may have more information.';
    Win32ErrorCodes.FRS_ERR_SYSVOL_POPULATE_TIMEOUT:
        Win32ErrorCodeDescription := 'The file replication service cannot populate the system volume because of an internal timeout. The event log may have more information.';
    Win32ErrorCodes.FRS_ERR_SYSVOL_IS_BUSY:
        Win32ErrorCodeDescription := 'The file replication service cannot process the request. The system volume is busy with a previous request.';
    Win32ErrorCodes.FRS_ERR_SYSVOL_DEMOTE:
        Win32ErrorCodeDescription := 'The file replication service cannot stop replicating the system volume because of an internal error. The event log may have more information.';
    Win32ErrorCodes.FRS_ERR_INVALID_SERVICE_PARAMETER:
        Win32ErrorCodeDescription := 'The file replication service detected an invalid parameter.';
    Win32ErrorCodes.ERROR_DS_NOT_INSTALLED:
        Win32ErrorCodeDescription := 'An error occurred while installing the directory service. For more information, see the event log.';
    Win32ErrorCodes.ERROR_DS_MEMBERSHIP_EVALUATED_LOCALLY:
        Win32ErrorCodeDescription := 'The directory service evaluated group memberships locally.';
    Win32ErrorCodes.ERROR_DS_NO_ATTRIBUTE_OR_VALUE:
        Win32ErrorCodeDescription :=
            'The specified directory service attribute or value does not exist.';
    Win32ErrorCodes.ERROR_DS_INVALID_ATTRIBUTE_SYNTAX:
        Win32ErrorCodeDescription :=
            'The attribute syntax specified to the directory service is invalid.';
    Win32ErrorCodes.ERROR_DS_ATTRIBUTE_TYPE_UNDEFINED:
        Win32ErrorCodeDescription :=
            'The attribute type specified to the directory service is not defined.';
    Win32ErrorCodes.ERROR_DS_ATTRIBUTE_OR_VALUE_EXISTS:
        Win32ErrorCodeDescription :=
            'The specified directory service attribute or value already exists.';
    Win32ErrorCodes.ERROR_DS_BUSY:
        Win32ErrorCodeDescription := 'The directory service is busy.';
    Win32ErrorCodes.ERROR_DS_UNAVAILABLE:
        Win32ErrorCodeDescription := 'The directory service is unavailable.';
    Win32ErrorCodes.ERROR_DS_NO_RIDS_ALLOCATED:
        Win32ErrorCodeDescription :=
            'The directory service was unable to allocate a relative identifier.';
    Win32ErrorCodes.ERROR_DS_NO_MORE_RIDS:
        Win32ErrorCodeDescription :=
